# B&R Automation Studio project NewPendant_NG4_11_05_25A (part 18)

```c
					/////////////////////////
					/////   Hardcoded Limits
					if(cfg->HeadCfg.OSC.Limits_Harcoded){

						curCalib->Points[CALIB_OSC_SFT_LIMIT].num = 4;
						curCalib->Points[CALIB_OSC_SFT_LIMIT].val[0] = 10.0;
						curCalib->Points[CALIB_OSC_SFT_LIMIT].val[1] = 75.0;
						curCalib->Points[CALIB_OSC_SFT_LIMIT].val[2] = curCalib->Points[i].val[0];
						curCalib->Points[CALIB_OSC_SFT_LIMIT].val[3] = curCalib->Points[i].val[1];
					}

					////////////////////////////////////////////////

				break;

			}

		}

		for(i=0 ; i < 1 ; i++){

			switch(i){

				case 0:

					strcpy(Process[PROC_GAS].Name , "GAS");
					GAS_Param_Set[i].pPrc = &Process[PROC_GAS];

					//GAS_Param_Set[i].pSensInput     = &Hardware[1].Inp[5];  //FourAxis Head
					GAS_Param_Set[i].pOutput		= &Hardware[1].Outp[4];

				break;

			}

		}

		for(i=0 ; i < 1; i++){

			switch(i){

				case 0:

					strcpy(Process[PROC_COOL].Name , "COOLANT");
					COOL_Param_Set[i].pPrc = &Process[PROC_COOL];

					COOL_Param_Set[i].pSensInput     = &Hardware[1].Inp[4];  //FourAxis Head
					COOL_Param_Set[i].pOutput		= &Hardware[1].Outp[6];

				break;

			}

		}

		for(i=0 ; i < 1; i++){

			switch(i){

				case 0:

					strcpy(Process[PROC_HW_PS].Name , "HW PS");
					HW_PS_Param_Set[i].pPrc = &Process[PROC_HW_PS];

					HW_PS_Param_Set[i].pCalibPoints		= &m->pCalib->Points[CALIB_HW_AMPS_CMD];
					HW_PS_Param_Set[i].rawCmdMax 		= 16383.0;
					HW_PS_Param_Set[i].AmpCMD_Max 		= 160.0;

					Process[PROC_HW_PS].Disable = 1;

				break;

			}

		}

		for(i=0 ; i < 2; i++){

			switch(i){

				case 0:

					strcpy(Process[PROC_WIRE_FEED].Name ,"WrFeed");
					strcpy(VectorStateMach[VECT_WF].Name ,"WrFeed#1");
					strcpy(VectorStateMach[VECT_WF_1].Name ,"WrFeed#2");

					WIRE_Param_Set[i].pPrc = &Process[PROC_WIRE_FEED];
					WIRE_Param_Set[i].pVect = &VectorStateMach[m->pCfg->HeadCfg.WF.VECT_A_Indx];
					WIRE_Param_Set[i].VectStateNum = 1;
					WIRE_Param_Set[i].Mode = 0;  // classic

					WIRE_Param_Set[i].pCalibPoints	= &m->pCalib->Points[CALIB_WF_SPEED_CMD];

				break;

				case 1:

					strcpy(Process[PROC_WIRE_PULSE].Name ,"WrPulse");
					strcpy(VectorStateMach[VECT_WP].Name ,"WrPulse#1");
					strcpy(VectorStateMach[VECT_WP_1].Name ,"WrPulse#2");

					WIRE_Param_Set[i].pPrc = &Process[PROC_WIRE_PULSE];
					WIRE_Param_Set[i].pVect = &VectorStateMach[m->pCfg->HeadCfg.WP.VECT_A_Indx];
					WIRE_Param_Set[i].VectStateNum = 1;

					WIRE_Param_Set[i].pCalibPoints	= &m->pCalib->Points[CALIB_WP_SPEED_CMD];

					Process[PROC_WIRE_PULSE].Disable = 1;

				break;

		}

		}

		for(i=0 ; i < 1; i++){

			switch(i){

				case 0:

					strcpy(Process[PROC_TVL].Name , "TVL");
					strcpy(VectorStateMach[VECT_TVL].Name , "TVL");

					TVL_ROT_Param_Set[i].pPrc = &Process[PROC_TVL];
					TVL_ROT_Param_Set[i].pVect = &VectorStateMach[VECT_TVL];
					TVL_ROT_Param_Set[i].VectStateNum = 1;

					TVL_ROT_Param_Set[i].VectModeForJog = vectSt_Mode_Volt;

					TVL_ROT_Param_Set[i].MaxSpeedJog = 24.0;

					TVL_ROT_Param_Set[i].TotalRescaleFactor = 1.0;
					TVL_ROT_Param_Set[i].pCalibPoints = &m->pCalib->Points[CALIB_TVL_SPEED_CMD];

					TVL_ROT_Param_Set[i].pTrackDia = &curCfg->Param[parTVL_TrackDia].val[0];
					TVL_ROT_Param_Set[i].pVelTolerance = &curCfg->Param[parTVL_SpeedTolerane].val[0];

					TVL_ROT_Param_Set[i].pEncoder = &AxisCh[TML_AX_TVL].curPos;
					TVL_ROT_Param_Set[i].pHomePos = &OLD_MTR_POS[TVL_ENC_HOME];
					TVL_ROT_Param_Set[i].EncPerTick = m->pCfg->HeadCfg.TVL.EncPerTick;
					TVL_ROT_Param_Set[i].EncDir = m->pCfg->HeadCfg.TVL.Enc_Dir;
					TVL_ROT_Param_Set[i].TicksAtHighVel = 3;

				break;

			}
		}

		for(i=0 ; i < 1 ; i++){

			switch(i){

				case 0:

					strcpy(Process[m->pCfg->HeadCfg.INDX.PROC_Indx].Name , "INDX");
					INDEX_Param_Set[i].pPrc = &Process[m->pCfg->HeadCfg.INDX.PROC_Indx];
					Process[m->pCfg->HeadCfg.INDX.PROC_Indx].Disable = 1;

				break;

			}

		}

	return 1;

}

DINT Configure_F_HEAD_HP_MINI_ENC(MASTER_typ * m,UINT headType){
int i;

CurCfg_typ *curCfg;
Cfg_typ *cfg;
CurCalib_typ *curCalib , *defaultCalib;

	if(!m)
		return;

	curCfg = (CurCfg_typ*)m->pCurCfg;
	cfg = (Cfg_typ*)m->pCfg;

	curCalib = m->pCalib;
	defaultCalib = m->pDefaultCalib;

	if(!curCfg || !cfg || !curCalib  || !defaultCalib)
		return;

	/*********************************************/
	/***   Hardware and Vectors *********************/

	TML_MTR_INST[m->pCfg->HeadCfg.TVL.TML_Indx ].pState = &VectorStateMach[m->pCfg->HeadCfg.TVL.VECT_Indx];

	TML_MTR_INST[m->pCfg->HeadCfg.AVC.TML_A_Indx ].pState = &VectorStateMach[m->pCfg->HeadCfg.AVC.VECT_A_Indx];
	TML_MTR_INST[m->pCfg->HeadCfg.AVC.TML_B_Indx ].pState = &VectorStateMach[m->pCfg->HeadCfg.AVC.VECT_B_Indx];

	TML_MTR_INST[m->pCfg->HeadCfg.OSC.TML_A_Indx ].pState = &VectorStateMach[m->pCfg->HeadCfg.OSC.VECT_A_Indx];
	TML_MTR_INST[m->pCfg->HeadCfg.OSC.TML_B_Indx ].pState = &VectorStateMach[m->pCfg->HeadCfg.OSC.VECT_B_Indx];

	DC_Mtr[m->pCfg->HeadCfg.WF.DC_A_Indx ].pState = &VectorStateMach[m->pCfg->HeadCfg.WF.VECT_A_Indx];
	DC_Mtr[m->pCfg->HeadCfg.WP.DC_A_Indx ].pState = &VectorStateMach[m->pCfg->HeadCfg.WP.VECT_A_Indx];
	DC_Mtr[m->pCfg->HeadCfg.WF.DC_B_Indx ].pState = &VectorStateMach[m->pCfg->HeadCfg.WF.VECT_B_Indx];
	DC_Mtr[m->pCfg->HeadCfg.WP.DC_B_Indx ].pState = &VectorStateMach[m->pCfg->HeadCfg.WP.VECT_B_Indx];

/*

	VectorStateMach[VECT_AVC].simul = 1;
	VectorStateMach[VECT_OSC].simul = 1;
	VectorStateMach[VECT_TVL].simul = 1;
	VectorStateMach[VECT_WF].simul = 1;
	VectorStateMach[VECT_WP].simul = 1;
	VectorStateMach[VECT_WF_1].simul = 1;
	VectorStateMach[VECT_WP_1].simul = 1;
		m->pCfg->HeadCfg.WF.VECT_A_Indx]
	DC_Mtr[DC_AX_WF].Disable = 1;
	DC_Mtr[DC_AX_WP].Disable = 1;
	DC_Mtr[DC_AX_WF_1].Disable = 1;
	DC_Mtr[DC_AX_WP_1].Disable = 1;

	TML_MTR_INST[TML_AX_AVC].Disable = 1;
	TML_MTR_INST[TML_AX_OSC].Disable = 1;
	TML_MTR_INST[TML_AX_TVL].Disable = 1;

	//Process[PROC_AVC].Disable = 1;
	Process[PROC_AVC].TestMode = 1;
*/
	Process[PROC_TVL].Disable = 0;
	Process[PROC_OSC].Disable = 0;
	Process[PROC_AVC].Disable = 0;
	Process[PROC_WIRE_FEED].Disable = 0;
	Process[PROC_WIRE_PULSE].Disable = 0;

	VectorStateMach[VECT_AVC].simul = 0;
	VectorStateMach[VECT_OSC].simul = 0;
	VectorStateMach[VECT_TVL].simul = 0;

	DC_Mtr[DC_AX_WF].Disable = 0;
	DC_Mtr[DC_AX_WP].Disable = 0;
	DC_Mtr[DC_AX_WF_1].Disable = 1;
	DC_Mtr[DC_AX_WP_1].Disable = 1;

	TML_MTR_INST[TML_AX_AVC].Disable = 0;
	TML_MTR_INST[TML_AX_OSC].Disable = 0;
	TML_MTR_INST[TML_AX_TVL].Disable = 0;

	/*********************************************************/
	/****   Phisical hardware configuration   ************************/

		for(i = 0 ; i < PROCESS_NUM; i++)
			strcpy(Process[i].Name , "spare");

		for(i = 0 ; i < VECTORS_NUM; i++)
			strcpy(VectorStateMach[i].Name , "spare");

		//////////////////////////////////////////////////////////////////////////////////
		// Wire Block
		for(i=0 ; i < 2; i++){

			switch(i){

				case 0:
					strcpy(Process[m->pCfg->HeadCfg.WB[i].PROC_Indx].Name , "WB_UD");
					strcpy(VectorStateMach[m->pCfg->HeadCfg.WB[i].VECT_Indx].Name , "WB_UD");

					WR_BLK_Param_Set[i].pPrc = &Process[m->pCfg->HeadCfg.WB[i].PROC_Indx];
					WR_BLK_Param_Set[i].pVect = &VectorStateMach[m->pCfg->HeadCfg.WB[i].VECT_Indx];
					WR_BLK_Param_Set[i].VectStateNum = 1;

					WR_BLK_Param_Set[i].MaxSpeedJog = 24.0;

					Gen_one = 1.0;
					WR_BLK_Param_Set[i].pJogSpeed = &Gen_one;

				break;

				case 1:
					strcpy(Process[m->pCfg->HeadCfg.WB[i].PROC_Indx].Name , "WB_LR");
					strcpy(VectorStateMach[m->pCfg->HeadCfg.WB[i].VECT_Indx].Name , "WB_LR");

					WR_BLK_Param_Set[i].pPrc = &Process[PROC_WB_LR];
					WR_BLK_Param_Set[i].pVect = &VectorStateMach[VECT_WB_LR];
					WR_BLK_Param_Set[i].VectStateNum = 1;

					WR_BLK_Param_Set[i].MaxSpeedJog = 24.0;

					Gen_one = 1.0;
					WR_BLK_Param_Set[i].pJogSpeed = &Gen_one;

				break;

			}

		}

		for(i = 0 ; i < DC2DIRMTR_NUM; i++){

			switch(i){

				case DC_WB_UD:

					strcpy(DC2DirMtr[i].Name , "WB_UD");
					DC2DirMtr[i].pState = &VectorStateMach[VECT_WB_UD];

					DC2DirMtr[i].Cfg.pQ1_output = &Hardware[1].Outp[12];
					DC2DirMtr[i].Cfg.pQ2_output = &Hardware[1].Outp[13];
					DC2DirMtr[i].Cfg.pQ3_output = &Hardware[1].Outp[14];
					DC2DirMtr[i].Cfg.pQ4_output = &Hardware[1].Outp[15];

					DC2DirMtr[i].Cfg.MtrDir = 1.0;

				break;

				case DC_WB_LR:

					strcpy(DC2DirMtr[i].Name , "WB_LR");
					DC2DirMtr[i].pState = &VectorStateMach[VECT_WB_LR];

					DC2DirMtr[i].Cfg.pQ1_output = &Hardware[1].Outp[16];
					DC2DirMtr[i].Cfg.pQ2_output = &Hardware[1].Outp[17];
					DC2DirMtr[i].Cfg.pQ3_output = &Hardware[1].Outp[18];
					DC2DirMtr[i].Cfg.pQ4_output = &Hardware[1].Outp[19];

					DC2DirMtr[i].Cfg.MtrDir = 1.0;

				break;

			}

		}
		/////////////////////////////////////////////////////////////////////////////////

		for(i = 0 ; i < GEN_MTR_NUM; i++){

			switch(i){

				case DC_AX_WF:
				case DC_AX_WF_1:

					switch(i){

						case DC_AX_WF:

							strcpy(DC_Mtr[i].Name , "DC WFeed#1");

							DC_Mtr[i].Cfg.mtr_dir = 1.0;

							if(ProjectConfig == project_US_Orbital) // US Orbital has B and /B swapped
								DC_Mtr[i].Cfg.enc_dir = -1.0;
							else
								DC_Mtr[i].Cfg.enc_dir = 1.0;

						break;

						case DC_AX_WF_1:

							strcpy(DC_Mtr[i].Name , "DC WFeed#2");

							//DC_Mtr[i].Cfg.mtr_dir = -1.0;
							DC_Mtr[i].Cfg.mtr_dir = 1.0;

							if(ProjectConfig == project_US_Orbital) // US Orbital has B and /B swapped
								DC_Mtr[i].Cfg.enc_dir = -1.0;
							else
								DC_Mtr[i].Cfg.enc_dir = 1.0;

						break;

					}

					//DC_Mtr[i].Cfg.units = 59.847340050885561192713356451475; // 0.75 " dia * 25.4 * PI
					DC_Mtr[i].Cfg.units = 2000 / 59.847340050885561192713356451475; // 2000 enc ticks / 0.75 " dia * 25.4 * PI
					DC_Mtr[i].Cfg.rev_scale = 66.0;	// Ratio gear box 66:1

					/* Parameters for PID controller */
					// To nowe
					DC_Mtr[i].msc.PIDParameters.Kp= 1.0;//0.4; //proportional gain / was 0.6
					//DC_Mtr[i].msc.PIDParameters.Kp= 0.1;//0.4; //proportional gain / was 0.6
					DC_Mtr[i].msc.PIDParameters.Tn= 0.1;//0.3.1; //intergral action time
					DC_Mtr[i].msc.PIDParameters.Kfbk = 0.01; //windup dampenin

					DC_Mtr[i].msc.PID.enable = 0;
					DC_Mtr[i].msc.PID.pPar = &DC_Mtr[i].msc.PIDParameters;
					DC_Mtr[i].msc.PID.request = 3; // Read parameters from PIDParameters
					DC_Mtr[i].msc.PIDParameters.Tv= 0; //derivative action time
					DC_Mtr[i].msc.PIDParameters.Y_max = 100.0;  //max manipulated variable %
					DC_Mtr[i].msc.PIDParameters.Y_min = -100.0; //min manipulated variable %

				break;

				case DC_AX_WP:
				case DC_AX_WP_1:

					switch(i){

						case DC_AX_WP:

							strcpy(DC_Mtr[i].Name , "DC WPulse#1");

							DC_Mtr[i].Cfg.mtr_dir = 1.0;

							if(ProjectConfig == project_US_Orbital) // US Orbital has B and /B swapped
								DC_Mtr[i].Cfg.enc_dir = -1.0;
							else
								DC_Mtr[i].Cfg.enc_dir = 1.0;

						break;

						case DC_AX_WP_1:

							strcpy(DC_Mtr[i].Name , "DC WPulse#2");

							DC_Mtr[i].Cfg.mtr_dir = 1.0;

							if(ProjectConfig == project_US_Orbital) // US Orbital has B and /B swapped
								DC_Mtr[i].Cfg.enc_dir = -1.0;
							else
								DC_Mtr[i].Cfg.enc_dir = 1.0;

						break;

					}

					//oryginalnie jest 2000 pulsow na obrot potem ratio on gear 4.8 : 1
					DC_Mtr[i].Cfg.units = 2000;
					DC_Mtr[i].Cfg.rev_scale = 4.8;// ratio on gear 4.8

					/* Parameters for PID controller */
					// To nowe
					DC_Mtr[i].msc.PIDParameters.Kp= 1.0;//0.4; //proportional gain / was 0.6
					//DC_Mtr[i].msc.PIDParameters.Kp= 0.1;//0.4; //proportional gain / was 0.6
					DC_Mtr[i].msc.PIDParameters.Tn= 0.1;//0.3.1; //intergral action time
					DC_Mtr[i].msc.PIDParameters.Kfbk = 0.01; //windup dampenin

					DC_Mtr[i].msc.PID.enable = 0;
					DC_Mtr[i].msc.PID.pPar = &DC_Mtr[i].msc.PIDParameters;
					DC_Mtr[i].msc.PID.request = 3; // Read parameters from PIDParameters
					DC_Mtr[i].msc.PIDParameters.Tv= 0; //derivative action time
					DC_Mtr[i].msc.PIDParameters.Y_max = 100.0;  //max manipulated variable %
					DC_Mtr[i].msc.PIDParameters.Y_min = -100.0; //min manipulated variable %

				break;

				default:

					strcpy(DC_Mtr[i].Name , "Spare ");

				break;

			}

			//CalcUnits(&DC_Mtr[i]);
			DC_Mtr[i].msc.kPos = (float)DC_Mtr[i].Cfg.units * DC_Mtr[i].Cfg.rev_scale;

		}

		/***********************************/

			for(i = 0 ; i < TML_SERVO_NUM ; i++){

				switch(i){

					// tml->_int.kPos = (tml->_cfg.units * tml->_cfg.rev_scale) / tml->_cfg.rev_motor;
					case TML_AX_AVC:

						strcpy(TML_MTR_INST[i].Name , "AVC");

						// Analog Feedback from REF
						TML_MTR_INST[i]._cfg.loopPeriod = 0.001;
						TML_MTR_INST[i]._cfg.units = 4095;
						TML_MTR_INST[i]._cfg.rev_motor = 1;
						TML_MTR_INST[i]._cfg.rev_scale = 1.0/5.0;
						TML_MTR_INST[i]._cfg.maxVel = 10.0; //1//6000 rpm
						TML_MTR_INST[i]._cfg.maxAcc = 100000.0;
						//TML_MTR_INST[i]._cfg.satpMax = 27853; // KPP bylo Stauration of proportional gain
						TML_MTR_INST[i]._cfg.satpMax = 32000; // KPP bylo Stauration of proportional gain
						TML_MTR_INST[i]._cfg.kppMax = 32000; // KPP bylo Stauration of proportional gain
						TML_MTR_INST[i]._cfg.kipMax = 200; // KPP bylo Stauration of proportional gain
						TML_MTR_INST[i]._cfg.absFbk = 0; // absolute value feedback

						TML_MTR_INST[i]._cfg.signFilter = curCfg->Param[parAVC_FbkFilter].val[0];

						if(ProjectConfig == project_US_Orbital){
							strcpy(TML_MTR_INST[i]._cfg.programName , "1423_AVC_FH_MINI_ENC_US.sw");
							TML_MTR_INST[i].ProgramVersion = ASC2UDINT("1423");
							TML_MTR_INST[i].FirmwareVersion = ASC2UDINT("6A2B");  //0x674B
							TML_MTR_INST[i]._cfg.Appl_ID_adr = 0x7FCF;

						}
						else{
							strcpy(TML_MTR_INST[i]._cfg.programName , "0423_AVC_FH_MINI_ENC.sw");
							TML_MTR_INST[i].ProgramVersion = ASC2UDINT("0423");
							TML_MTR_INST[i].FirmwareVersion = ASC2UDINT("674C");  //0x674C
						}

						//TML_MTR_INST[i]._cfg.sftLimitPos = 1000.0;
						//TML_MTR_INST[i]._cfg.sftLimitNeg = -1000.0;

					break;

					case TML_AX_OSC:

						strcpy(TML_MTR_INST[i].Name , "OSC");

						if(ProjectConfig == project_US_Orbital){
							strcpy(TML_MTR_INST[i]._cfg.programName , "1412_OSC_FH_MINI_ENC_US.sw");
							TML_MTR_INST[i].ProgramVersion = ASC2UDINT("1412");
							TML_MTR_INST[i].FirmwareVersion = ASC2UDINT("6A2B");  //0x674B
							TML_MTR_INST[i]._cfg.Appl_ID_adr = 0x7FCF;

						}
						else{
							strcpy(TML_MTR_INST[i]._cfg.programName , "0412_OSC_FH_MINI_ENC.sw");
							TML_MTR_INST[i].ProgramVersion = ASC2UDINT("0412");
							TML_MTR_INST[i].FirmwareVersion = ASC2UDINT("674C");  //0x674C
						}

						TML_MTR_INST[i]._cfg.loopPeriod = 0.001;
						TML_MTR_INST[i]._cfg.absFbk = 0; // value fom APOS which is analog Ref
						TML_MTR_INST[i]._cfg.units = 4096.0 ;
						TML_MTR_INST[i]._cfg.rev_motor = 1;
						TML_MTR_INST[i]._cfg.rev_scale = 1.0 / 80.0;  // this comes from experiment
						//TML_MTR_INST[i]._cfg.rev_scale = 1.0 / 56.0; // this comes from drawings
						TML_MTR_INST[i]._cfg.maxVel = 100.0;
						TML_MTR_INST[i]._cfg.maxAcc = 100.0;

						TML_MTR_INST[i]._cfg.AnalLimitPos = 3900;
						TML_MTR_INST[i]._cfg.AnalLimitNeg = 100;

					break;

					case TML_AX_TVL:

						strcpy(TML_MTR_INST[i].Name , "TVL");

						/// Deferent TML programs
						// Back EMF
						TML_MTR_INST[i]._cfg.loopPeriod = 0.001;

						if(ProjectConfig == project_US_Orbital){
							strcpy(TML_MTR_INST[i]._cfg.programName , "1411_TVL_FH_MINI_ENC_US.sw");
							TML_MTR_INST[i].ProgramVersion = ASC2UDINT("1411");
							TML_MTR_INST[i].FirmwareVersion = ASC2UDINT("6A2B");  //0x674B
							TML_MTR_INST[i]._cfg.Appl_ID_adr = 0x7FCF;

						}
						else{
							strcpy(TML_MTR_INST[i]._cfg.programName , "0411_TVL_FH_MINI_ENC.sw");
							TML_MTR_INST[i].ProgramVersion = ASC2UDINT("0411");
							TML_MTR_INST[i].FirmwareVersion = ASC2UDINT("674C");  //0x674C
						}

						TML_MTR_INST[i]._cfg.units =  1000; //  to jest tyle ile z max speed TML EREF
						TML_MTR_INST[i]._cfg.rev_scale = -1920.0;
						TML_MTR_INST[i]._cfg.rev_motor = 1.0 ;
						TML_MTR_INST[i]._cfg.maxVel =  10.0; // mm/s
						TML_MTR_INST[i]._cfg.maxAcc = 100.0;
						TML_MTR_INST[i]._cfg.absFbk = 0; // non absolute value feedback , remember last value before drive reset

					break;

					default:

						xsprintf(TML_MTR_INST[i].Name, "Spare %d", i );
						TML_MTR_INST[i].pState = 0;

					break;

				}

			TML_MTR_INST[i].xCMD = TML_RESTART;

		}

		TML_mgr[0].hrdw[0].AxisNum = 3;
		TML_mgr[0].hrdw[1].AxisNum = 0;

		TML_mgr[0].pAxis[0] = &AxisCh[0];
		TML_mgr[0].pAxis[1] = 0;
		//TML_mgr[0].pAxis[1] = &AxisCh[TML_mgr[0].hrdw[0].AxisNum];

		TML_mgr[0].pTML[0] = &TML_MTR_INST[0];
		TML_mgr[0].pTML[1] = 0;
		//TML_mgr[0].pTML[1] = &TML_MTR_INST[TML_mgr[0].hrdw[0].AxisNum];

		AxisCh[TML_AX_TVL].AxisID	= 1;
		AxisCh[TML_AX_OSC].AxisID 	= 2;
		AxisCh[TML_AX_AVC].AxisID 	= 3;

		/**************************************/
		/****   Process   ************************/

		// Lincoln Power Supply
		for(i=0 ; i < 1; i++){

			switch(i){

				case 0:

					strcpy(Process[PROC_TIG_PS].Name , "TIG PS");
					PS_Param_Set[i].pPrc = &Process[PROC_TIG_PS];

					PS_Param_Set[i].pCalibPoints		= &m->pCalib->Points[CALIB_TIG_AMPS_CMD];
					//PS_Param_Set[i].rawCmdMax			= 26170; // //
					//PS_Param_Set[i].AmpCMD_Max			= 500.0; // 62.5 amp / 1 V
					PS_Param_Set[i].rawCmdMax			= 32767;
					PS_Param_Set[i].AmpCMD_Max			= 627.0;

					PS_Param_Set[i].pArcLinkRobot   = (UDINT)&ArcLink.robot;

				break;

			}

		}

		for(i=0 ; i < 1 ; i++){

			switch(i){

				case 0:

					strcpy(Process[PROC_AVC].Name , "AVC");

					strcpy(VectorStateMach[VECT_AVC].Name , "AVC");

					AVC_Param_Set[i].pPrc = &Process[PROC_AVC];
					AVC_Param_Set[i].pVect = &VectorStateMach[VECT_AVC];
					AVC_Param_Set[i].VectStateNum = 1;
					AVC_Param_Set[i].Mode = 0;

					AVC_Param_Set[i].MaxSpeedJog = 24.0;

					m->pCalib->Points[CALIB_TIG_VOLT_FBK].num = 10;
					AVC_Param_Set[i].pCalibPoints		= &m->pCalib->Points[CALIB_TIG_VOLT_FBK];

				break;

			}
		}

		for(i=0 ; i < 1 ; i++){

			switch(i){

				case 0:

					strcpy(Process[PROC_OSC].Name , "OSC");
					strcpy(VectorStateMach[VECT_OSC].Name , "OSC");

					OSC_TML_Param_Set[i].pPrc = &Process[PROC_OSC];
					OSC_TML_Param_Set[i].pVect = &VectorStateMach[VECT_OSC];
					OSC_TML_Param_Set[i].VectStateNum = 1;
					OSC_TML_Param_Set[i].pTML = &TML_MTR_INST[TML_AX_OSC] ;

					OSC_TML_Param_Set[i].Mode = 0;

					////  New Oscillation concept - BEMF
					OSC_TML_Param_Set[i].mm2ticks = TML_MTR_INST[TML_AX_OSC]._cfg.units * TML_MTR_INST[TML_AX_OSC]._cfg.rev_scale;
			 		OSC_TML_Param_Set[i].SpeedFactor = 410;
					//OSC_TML_Param_Set[i].MaxOscAmpl = 1.0 * 25.4;
					OSC_TML_Param_Set[i].MaxOscAmpl = 0.0;

					/////////////////////////
					/////   Hardcoded Limits
					if(cfg->HeadCfg.OSC.Limits_Harcoded){

						curCalib->Points[CALIB_OSC_SFT_LIMIT].num = 4;
						curCalib->Points[CALIB_OSC_SFT_LIMIT].val[0] = 10.0;
						curCalib->Points[CALIB_OSC_SFT_LIMIT].val[1] = 75.0;
						curCalib->Points[CALIB_OSC_SFT_LIMIT].val[2] = curCalib->Points[i].val[0];
						curCalib->Points[CALIB_OSC_SFT_LIMIT].val[3] = curCalib->Points[i].val[1];
					}

					////////////////////////////////////////////////

				break;

			}

		}

		for(i=0 ; i < 1 ; i++){

			switch(i){

				case 0:

					strcpy(Process[PROC_GAS].Name , "GAS");
					GAS_Param_Set[i].pPrc = &Process[PROC_GAS];

					//GAS_Param_Set[i].pSensInput     = &Hardware[1].Inp[5];  //FourAxis Head
					GAS_Param_Set[i].pOutput		= &Hardware[1].Outp[4];

				break;

			}

		}

		for(i=0 ; i < 1; i++){

			switch(i){

				case 0:

					strcpy(Process[PROC_COOL].Name , "COOLANT");
					COOL_Param_Set[i].pPrc = &Process[PROC_COOL];

					COOL_Param_Set[i].pSensInput     = &Hardware[1].Inp[4];  //FourAxis Head
					COOL_Param_Set[i].pOutput		= &Hardware[1].Outp[6];

				break;

			}

		}

		for(i=0 ; i < 1; i++){

			switch(i){

				case 0:

					strcpy(Process[PROC_HW_PS].Name , "HW PS");
					HW_PS_Param_Set[i].pPrc = &Process[PROC_HW_PS];

					HW_PS_Param_Set[i].pCalibPoints		= &m->pCalib->Points[CALIB_HW_AMPS_CMD];
					HW_PS_Param_Set[i].rawCmdMax 		= 16383.0;
					HW_PS_Param_Set[i].AmpCMD_Max 		= 160.0;

				break;

			}

		}

		for(i=0 ; i < 2; i++){

			switch(i){

				case 0:

					strcpy(Process[PROC_WIRE_FEED].Name ,"WrFeed");
					strcpy(VectorStateMach[VECT_WF].Name ,"WrFeed#1");
					strcpy(VectorStateMach[VECT_WF_1].Name ,"WrFeed#2");

					WIRE_Param_Set[i].pPrc = &Process[PROC_WIRE_FEED];
					WIRE_Param_Set[i].pVect = &VectorStateMach[m->pCfg->HeadCfg.WF.VECT_A_Indx];
					WIRE_Param_Set[i].VectStateNum = 1;
					WIRE_Param_Set[i].Mode = 0;  // classic

					WIRE_Param_Set[i].pCalibPoints	= &m->pCalib->Points[CALIB_WF_SPEED_CMD];

				break;

				case 1:

					strcpy(Process[PROC_WIRE_PULSE].Name ,"WrPulse");
					strcpy(VectorStateMach[VECT_WP].Name ,"WrPulse#1");
					strcpy(VectorStateMach[VECT_WP_1].Name ,"WrPulse#2");

					WIRE_Param_Set[i].pPrc = &Process[PROC_WIRE_PULSE];
					WIRE_Param_Set[i].pVect = &VectorStateMach[m->pCfg->HeadCfg.WP.VECT_A_Indx];
					WIRE_Param_Set[i].VectStateNum = 1;

					WIRE_Param_Set[i].pCalibPoints	= &m->pCalib->Points[CALIB_WP_SPEED_CMD];

				break;

		}

		}

		for(i=0 ; i < 1; i++){

			switch(i){

				case 0:

					strcpy(Process[PROC_TVL].Name , "TVL");
					strcpy(VectorStateMach[VECT_TVL].Name , "TVL");

					TVL_ROT_Param_Set[i].pPrc = &Process[PROC_TVL];
					TVL_ROT_Param_Set[i].pVect = &VectorStateMach[VECT_TVL];
					TVL_ROT_Param_Set[i].VectStateNum = 1;

					TVL_ROT_Param_Set[i].VectModeForJog = vectSt_Mode_Volt;

					TVL_ROT_Param_Set[i].MaxSpeedJog = 24.0;

					TVL_ROT_Param_Set[i].TotalRescaleFactor = 1.0;
					TVL_ROT_Param_Set[i].pCalibPoints = &m->pCalib->Points[CALIB_TVL_SPEED_CMD];

					TVL_ROT_Param_Set[i].pTrackDia = &curCfg->Param[parTVL_TrackDia].val[0];
					TVL_ROT_Param_Set[i].pVelTolerance = &curCfg->Param[parTVL_SpeedTolerane].val[0];

					TVL_ROT_Param_Set[i].pEncoder = &AxisCh[TML_AX_TVL].curPos;
					TVL_ROT_Param_Set[i].pHomePos = &OLD_MTR_POS[TVL_ENC_HOME];
					TVL_ROT_Param_Set[i].EncPerTick = m->pCfg->HeadCfg.TVL.EncPerTick;
					TVL_ROT_Param_Set[i].EncDir = m->pCfg->HeadCfg.TVL.Enc_Dir;
					TVL_ROT_Param_Set[i].TicksAtHighVel = 3;

				break;

			}
		}

		for(i=0 ; i < 1 ; i++){

			switch(i){

				case 0:

					strcpy(Process[m->pCfg->HeadCfg.INDX.PROC_Indx].Name , "INDX");
					INDEX_Param_Set[i].pPrc = &Process[m->pCfg->HeadCfg.INDX.PROC_Indx];
					Process[m->pCfg->HeadCfg.INDX.PROC_Indx].Disable = 1;

				break;

			}

		}

	return 1;

}

DINT Configure_D_HEAD_HP(MASTER_typ * m,UINT headType){
int i;

CurCfg_typ *curCfg;
Cfg_typ *cfg;
CurCalib_typ *curCalib , *defaultCalib;

	if(!m)
		return;

	curCfg = (CurCfg_typ*)m->pCurCfg;
	cfg = (Cfg_typ*)m->pCfg;

	curCalib = m->pCalib;
	defaultCalib = m->pDefaultCalib;

	if(!curCfg || !cfg || !curCalib  || !defaultCalib)
		return;

	/*********************************************/
	/***   Hardware and Vectors *********************/

	TML_MTR_INST[m->pCfg->HeadCfg.TVL.TML_Indx ].pState = &VectorStateMach[m->pCfg->HeadCfg.TVL.VECT_Indx];

	TML_MTR_INST[m->pCfg->HeadCfg.AVC.TML_A_Indx ].pState = &VectorStateMach[m->pCfg->HeadCfg.AVC.VECT_A_Indx];
	TML_MTR_INST[m->pCfg->HeadCfg.AVC.TML_B_Indx ].pState = &VectorStateMach[m->pCfg->HeadCfg.AVC.VECT_B_Indx];

	TML_MTR_INST[m->pCfg->HeadCfg.OSC.TML_A_Indx ].pState = &VectorStateMach[m->pCfg->HeadCfg.OSC.VECT_A_Indx];
	TML_MTR_INST[m->pCfg->HeadCfg.OSC.TML_B_Indx ].pState = &VectorStateMach[m->pCfg->HeadCfg.OSC.VECT_B_Indx];

	DC_Mtr[m->pCfg->HeadCfg.WF.DC_A_Indx ].pState = &VectorStateMach[m->pCfg->HeadCfg.WF.VECT_A_Indx];
	DC_Mtr[m->pCfg->HeadCfg.WP.DC_A_Indx ].pState = &VectorStateMach[m->pCfg->HeadCfg.WP.VECT_A_Indx];
	DC_Mtr[m->pCfg->HeadCfg.WF.DC_B_Indx ].pState = &VectorStateMach[m->pCfg->HeadCfg.WF.VECT_B_Indx];
	DC_Mtr[m->pCfg->HeadCfg.WP.DC_B_Indx ].pState = &VectorStateMach[m->pCfg->HeadCfg.WP.VECT_B_Indx];

/*

	VectorStateMach[VECT_AVC].simul = 1;
	VectorStateMach[VECT_OSC].simul = 1;
	VectorStateMach[VECT_TVL].simul = 1;
	VectorStateMach[VECT_WF].simul = 1;
	VectorStateMach[VECT_WP].simul = 1;
	VectorStateMach[VECT_WF_1].simul = 1;
	VectorStateMach[VECT_WP_1].simul = 1;
		m->pCfg->HeadCfg.WF.VECT_A_Indx]
	DC_Mtr[DC_AX_WF].Disable = 1;
	DC_Mtr[DC_AX_WP].Disable = 1;
	DC_Mtr[DC_AX_WF_1].Disable = 1;
	DC_Mtr[DC_AX_WP_1].Disable = 1;

	TML_MTR_INST[TML_AX_AVC].Disable = 1;
	TML_MTR_INST[TML_AX_OSC].Disable = 1;
	TML_MTR_INST[TML_AX_TVL].Disable = 1;

	//Process[PROC_AVC].Disable = 1;
	Process[PROC_AVC].TestMode = 1;
*/
	Process[PROC_TVL].Disable = 0;
	Process[PROC_OSC].Disable = 0;
	Process[PROC_AVC].Disable = 0;
	Process[PROC_WIRE_FEED].Disable = 0;
	Process[PROC_WIRE_PULSE].Disable = 0;

	VectorStateMach[VECT_AVC].simul = 0;
	VectorStateMach[VECT_OSC].simul = 0;
	VectorStateMach[VECT_TVL].simul = 0;

	DC_Mtr[DC_AX_WF].Disable = 0;
	DC_Mtr[DC_AX_WP].Disable = 0;
	DC_Mtr[DC_AX_WF_1].Disable = 1;
	DC_Mtr[DC_AX_WP_1].Disable = 1;

	TML_MTR_INST[TML_AX_AVC].Disable = 0;
	TML_MTR_INST[TML_AX_OSC].Disable = 0;
	TML_MTR_INST[TML_AX_TVL].Disable = 0;

	/*********************************************************/
	/****   Phisical hardware configuration   ************************/

		for(i = 0 ; i < PROCESS_NUM; i++)
			strcpy(Process[i].Name , "spare");

		for(i = 0 ; i < VECTORS_NUM; i++)
			strcpy(VectorStateMach[i].Name , "spare");

		//////////////////////////////////////////////////////////////////////////////////
		// Wire Block
		for(i=0 ; i < 2; i++){

			switch(i){

				case 0:
					strcpy(Process[m->pCfg->HeadCfg.WB[i].PROC_Indx].Name , "WB_UD");
					strcpy(VectorStateMach[m->pCfg->HeadCfg.WB[i].VECT_Indx].Name , "WB_UD");

					WR_BLK_Param_Set[i].pPrc = &Process[m->pCfg->HeadCfg.WB[i].PROC_Indx];
					WR_BLK_Param_Set[i].pVect = &VectorStateMach[m->pCfg->HeadCfg.WB[i].VECT_Indx];
					WR_BLK_Param_Set[i].VectStateNum = 1;

					WR_BLK_Param_Set[i].MaxSpeedJog = 24.0;

					Gen_one = 1.0;
					WR_BLK_Param_Set[i].pJogSpeed = &Gen_one;

				break;

				case 1:
					strcpy(Process[m->pCfg->HeadCfg.WB[i].PROC_Indx].Name , "WB_LR");
					strcpy(VectorStateMach[m->pCfg->HeadCfg.WB[i].VECT_Indx].Name , "WB_LR");

					WR_BLK_Param_Set[i].pPrc = &Process[PROC_WB_LR];
					WR_BLK_Param_Set[i].pVect = &VectorStateMach[VECT_WB_LR];
					WR_BLK_Param_Set[i].VectStateNum = 1;

					WR_BLK_Param_Set[i].MaxSpeedJog = 24.0;

					Gen_one = 1.0;
					WR_BLK_Param_Set[i].pJogSpeed = &Gen_one;

				break;

			}

		}

		for(i = 0 ; i < DC2DIRMTR_NUM; i++){

			switch(i){

				case DC_WB_UD:

					strcpy(DC2DirMtr[i].Name , "WB_UD");
					DC2DirMtr[i].pState = &VectorStateMach[VECT_WB_UD];

					DC2DirMtr[i].Cfg.pQ1_output = &Hardware[1].Outp[12];
					DC2DirMtr[i].Cfg.pQ2_output = &Hardware[1].Outp[13];
					DC2DirMtr[i].Cfg.pQ3_output = &Hardware[1].Outp[14];
					DC2DirMtr[i].Cfg.pQ4_output = &Hardware[1].Outp[15];

					DC2DirMtr[i].Cfg.MtrDir = 1.0;

				break;

				case DC_WB_LR:

					strcpy(DC2DirMtr[i].Name , "WB_LR");
					DC2DirMtr[i].pState = &VectorStateMach[VECT_WB_LR];

					DC2DirMtr[i].Cfg.pQ1_output = &Hardware[1].Outp[16];
					DC2DirMtr[i].Cfg.pQ2_output = &Hardware[1].Outp[17];
					DC2DirMtr[i].Cfg.pQ3_output = &Hardware[1].Outp[18];
					DC2DirMtr[i].Cfg.pQ4_output = &Hardware[1].Outp[19];

					DC2DirMtr[i].Cfg.MtrDir = 1.0;

				break;

			}

		}
		/////////////////////////////////////////////////////////////////////////////////

		for(i = 0 ; i < GEN_MTR_NUM; i++){

			switch(i){

				case DC_AX_WF:
				case DC_AX_WF_1:

					switch(i){

						case DC_AX_WF:

							strcpy(DC_Mtr[i].Name , "DC WFeed#1");

							DC_Mtr[i].Cfg.mtr_dir = 1.0;

							if(ProjectConfig == project_US_Orbital) // US Orbital has B and /B swapped
								DC_Mtr[i].Cfg.enc_dir = -1.0;
							else
								DC_Mtr[i].Cfg.enc_dir = 1.0;

						break;

						case DC_AX_WF_1:

							strcpy(DC_Mtr[i].Name , "DC WFeed#2");

							//DC_Mtr[i].Cfg.mtr_dir = -1.0;
							DC_Mtr[i].Cfg.mtr_dir = 1.0;

							if(ProjectConfig == project_US_Orbital) // US Orbital has B and /B swapped
								DC_Mtr[i].Cfg.enc_dir = -1.0;
							else
								DC_Mtr[i].Cfg.enc_dir = 1.0;

						break;

					}

					//DC_Mtr[i].Cfg.units = 59.847340050885561192713356451475; // 0.75 " dia * 25.4 * PI
					DC_Mtr[i].Cfg.units = 2000 / 59.847340050885561192713356451475; // 2000 enc ticks / 0.75 " dia * 25.4 * PI
					DC_Mtr[i].Cfg.rev_scale = 66.0;	// Ratio gear box 66:1

					/* Parameters for PID controller */
					// To nowe
					DC_Mtr[i].msc.PIDParameters.Kp= 1.0;//0.4; //proportional gain / was 0.6
					//DC_Mtr[i].msc.PIDParameters.Kp= 0.1;//0.4; //proportional gain / was 0.6
					DC_Mtr[i].msc.PIDParameters.Tn= 0.1;//0.3.1; //intergral action time
					DC_Mtr[i].msc.PIDParameters.Kfbk = 0.01; //windup dampenin

					DC_Mtr[i].msc.PID.enable = 0;
					DC_Mtr[i].msc.PID.pPar = &DC_Mtr[i].msc.PIDParameters;
					DC_Mtr[i].msc.PID.request = 3; // Read parameters from PIDParameters
					DC_Mtr[i].msc.PIDParameters.Tv= 0; //derivative action time
					DC_Mtr[i].msc.PIDParameters.Y_max = 100.0;  //max manipulated variable %
					DC_Mtr[i].msc.PIDParameters.Y_min = -100.0; //min manipulated variable %

				break;

				case DC_AX_WP:
				case DC_AX_WP_1:

					switch(i){

						case DC_AX_WP:

							strcpy(DC_Mtr[i].Name , "DC WPulse#1");

							DC_Mtr[i].Cfg.mtr_dir = 1.0;

							if(ProjectConfig == project_US_Orbital) // US Orbital has B and /B swapped
								DC_Mtr[i].Cfg.enc_dir = -1.0;
							else
								DC_Mtr[i].Cfg.enc_dir = 1.0;

						break;

						case DC_AX_WP_1:

							strcpy(DC_Mtr[i].Name , "DC WPulse#2");

							DC_Mtr[i].Cfg.mtr_dir = 1.0;

							if(ProjectConfig == project_US_Orbital) // US Orbital has B and /B swapped
								DC_Mtr[i].Cfg.enc_dir = -1.0;
							else
								DC_Mtr[i].Cfg.enc_dir = 1.0;

						break;

					}

					//oryginalnie jest 2000 pulsow na obrot potem ratio on gear 4.8 : 1
					DC_Mtr[i].Cfg.units = 2000;
					DC_Mtr[i].Cfg.rev_scale = 4.8;// ratio on gear 4.8

					/* Parameters for PID controller */
					// To nowe
					DC_Mtr[i].msc.PIDParameters.Kp= 1.0;//0.4; //proportional gain / was 0.6
					//DC_Mtr[i].msc.PIDParameters.Kp= 0.1;//0.4; //proportional gain / was 0.6
					DC_Mtr[i].msc.PIDParameters.Tn= 0.1;//0.3.1; //intergral action time
					DC_Mtr[i].msc.PIDParameters.Kfbk = 0.01; //windup dampenin

					DC_Mtr[i].msc.PID.enable = 0;
					DC_Mtr[i].msc.PID.pPar = &DC_Mtr[i].msc.PIDParameters;
					DC_Mtr[i].msc.PID.request = 3; // Read parameters from PIDParameters
					DC_Mtr[i].msc.PIDParameters.Tv= 0; //derivative action time
					DC_Mtr[i].msc.PIDParameters.Y_max = 100.0;  //max manipulated variable %
					DC_Mtr[i].msc.PIDParameters.Y_min = -100.0; //min manipulated variable %

				break;

				default:

					strcpy(DC_Mtr[i].Name , "Spare ");

				break;

			}

			//CalcUnits(&DC_Mtr[i]);
			DC_Mtr[i].msc.kPos = (float)DC_Mtr[i].Cfg.units * DC_Mtr[i].Cfg.rev_scale;

		}

		/***********************************/

			for(i = 0 ; i < TML_SERVO_NUM ; i++){

				switch(i){

					// tml->_int.kPos = (tml->_cfg.units * tml->_cfg.rev_scale) / tml->_cfg.rev_motor;
					case TML_AX_AVC:

						strcpy(TML_MTR_INST[i].Name , "AVC");

						// Analog Feedback from REF
						TML_MTR_INST[i]._cfg.loopPeriod = 0.001;
						TML_MTR_INST[i]._cfg.units = 4095;
						TML_MTR_INST[i]._cfg.rev_motor = -1;
						TML_MTR_INST[i]._cfg.rev_scale = 1.0/5.0;
						TML_MTR_INST[i]._cfg.maxVel = 10.0; //1//6000 rpm
						TML_MTR_INST[i]._cfg.maxAcc = 100000.0;
						//TML_MTR_INST[i]._cfg.satpMax = 27853; // KPP bylo Stauration of proportional gain
						TML_MTR_INST[i]._cfg.satpMax = 32000; // KPP bylo Stauration of proportional gain
						TML_MTR_INST[i]._cfg.kppMax = 32000; // KPP bylo Stauration of proportional gain
						TML_MTR_INST[i]._cfg.kipMax = 200; // KPP bylo Stauration of proportional gain
						TML_MTR_INST[i]._cfg.absFbk = 0; // absolute value feedback

						TML_MTR_INST[i]._cfg.signFilter = curCfg->Param[parAVC_FbkFilter].val[0];

						if(ProjectConfig == project_US_Orbital){

							strcpy(TML_MTR_INST[i]._cfg.programName , "1423_AVC_FH_MINI_ENC_US.sw");
							TML_MTR_INST[i].ProgramVersion = ASC2UDINT("1423");
							TML_MTR_INST[i].FirmwareVersion = ASC2UDINT("6A2B");  //0x674B
							TML_MTR_INST[i]._cfg.Appl_ID_adr = 0x7FCF;

						}
						else{
							strcpy(TML_MTR_INST[i]._cfg.programName , "0423_AVC_FH_MINI_ENC.sw");
							TML_MTR_INST[i].ProgramVersion = ASC2UDINT("0423");
							TML_MTR_INST[i].FirmwareVersion = ASC2UDINT("674C");  //0x674C
						}

						//TML_MTR_INST[i]._cfg.sftLimitPos = 1000.0;
						//TML_MTR_INST[i]._cfg.sftLimitNeg = -1000.0;

					break;

					case TML_AX_OSC:

						strcpy(TML_MTR_INST[i].Name , "OSC");

						if(ProjectConfig == project_US_Orbital){

							/*
							strcpy(TML_MTR_INST[i]._cfg.programName , "1412_OSC_FH_MINI_ENC_US.sw");
							TML_MTR_INST[i].ProgramVersion = ASC2UDINT("1412");
							TML_MTR_INST[i].FirmwareVersion = ASC2UDINT("6A2B");  //0x674B
							TML_MTR_INST[i]._cfg.Appl_ID_adr = 0x7FCF;
							*/

							// New Osc Mode -  11;
							strcpy(TML_MTR_INST[i]._cfg.programName , "2512_OSC_D_HEAD_US.sw");
							TML_MTR_INST[i].ProgramVersion = ASC2UDINT("2512");
							TML_MTR_INST[i].FirmwareVersion = ASC2UDINT("6A2B");  //0x674B
							TML_MTR_INST[i]._cfg.Appl_ID_adr = 0x7FCF;

						}
						else{
							strcpy(TML_MTR_INST[i]._cfg.programName , "0412_OSC_FH_MINI_ENC.sw");
							TML_MTR_INST[i].ProgramVersion = ASC2UDINT("0412");
							TML_MTR_INST[i].FirmwareVersion = ASC2UDINT("674C");  //0x674C
						}

						TML_MTR_INST[i]._cfg.loopPeriod = 0.001;
						TML_MTR_INST[i]._cfg.absFbk = 0; // value fom APOS which is analog Ref
						TML_MTR_INST[i]._cfg.units = 4096.0 ;
						TML_MTR_INST[i]._cfg.rev_motor = 1;
						TML_MTR_INST[i]._cfg.rev_scale = 0.0375;  // this comes from experiment
						//TML_MTR_INST[i]._cfg.rev_scale = 1.0 / 56.0; // this comes from drawings
						TML_MTR_INST[i]._cfg.maxVel = 100.0;
						TML_MTR_INST[i]._cfg.maxAcc = 100.0;

						TML_MTR_INST[i]._cfg.AnalLimitPos = 3900;
						TML_MTR_INST[i]._cfg.AnalLimitNeg = 100;

					break;

					case TML_AX_TVL:

						strcpy(TML_MTR_INST[i].Name , "TVL");

						/// Deferent TML programs
						// Back EMF
						TML_MTR_INST[i]._cfg.loopPeriod = 0.001;

						if(ProjectConfig == project_US_Orbital){
							strcpy(TML_MTR_INST[i]._cfg.programName , "2511_TVL_D_HEAD_US.sw");
							TML_MTR_INST[i].ProgramVersion = ASC2UDINT("2511");
							TML_MTR_INST[i].FirmwareVersion = ASC2UDINT("6A2B");  //0x674B
							TML_MTR_INST[i]._cfg.Appl_ID_adr = 0x7FCF;

						}
						else{
							strcpy(TML_MTR_INST[i]._cfg.programName , "0411_TVL_FH_MINI_ENC.sw");
							TML_MTR_INST[i].ProgramVersion = ASC2UDINT("0411");
							TML_MTR_INST[i].FirmwareVersion = ASC2UDINT("674C");  //0x674C
						}

						TML_MTR_INST[i]._cfg.units =  1000; //  to jest tyle ile z max speed TML EREF
						//TML_MTR_INST[i]._cfg.rev_scale = -1920.0;
						TML_MTR_INST[i]._cfg.rev_scale =4000.0;
						TML_MTR_INST[i]._cfg.rev_motor = 1.0 ;
						TML_MTR_INST[i]._cfg.maxVel =  4; // mm/s
						TML_MTR_INST[i]._cfg.maxAcc = 100.0;
						TML_MTR_INST[i]._cfg.absFbk = 0; // non absolute value feedback , remember last value before drive reset

					break;

					default:

						xsprintf(TML_MTR_INST[i].Name, "Spare %d", i );
						TML_MTR_INST[i].pState = 0;

					break;

				}

			TML_MTR_INST[i].xCMD = TML_RESTART;

		}

		TML_mgr[0].hrdw[0].AxisNum = 3;
		TML_mgr[0].hrdw[1].AxisNum = 0;

		TML_mgr[0].pAxis[0] = &AxisCh[0];
		TML_mgr[0].pAxis[1] = 0;
		//TML_mgr[0].pAxis[1] = &AxisCh[TML_mgr[0].hrdw[0].AxisNum];

		TML_mgr[0].pTML[0] = &TML_MTR_INST[0];
		TML_mgr[0].pTML[1] = 0;
		//TML_mgr[0].pTML[1] = &TML_MTR_INST[TML_mgr[0].hrdw[0].AxisNum];

		AxisCh[TML_AX_TVL].AxisID	= 1;
		AxisCh[TML_AX_OSC].AxisID 	= 2;
		AxisCh[TML_AX_AVC].AxisID 	= 3;

		/**************************************/
		/****   Process   ************************/

		// Lincoln Power Supply
		for(i=0 ; i < 1; i++){

			switch(i){

				case 0:

					strcpy(Process[PROC_TIG_PS].Name , "TIG PS");
					PS_Param_Set[i].pPrc = &Process[PROC_TIG_PS];

					PS_Param_Set[i].pCalibPoints		= &m->pCalib->Points[CALIB_TIG_AMPS_CMD];
					//PS_Param_Set[i].rawCmdMax			= 26170; // //
					//PS_Param_Set[i].AmpCMD_Max			= 500.0; // 62.5 amp / 1 V
					PS_Param_Set[i].rawCmdMax			= 32767;
					PS_Param_Set[i].AmpCMD_Max			= 627.0;

					PS_Param_Set[i].pArcLinkRobot   = (UDINT)&ArcLink.robot;

				break;

			}

		}

		for(i=0 ; i < 1 ; i++){

			switch(i){

				case 0:

					strcpy(Process[PROC_AVC].Name , "AVC");

					strcpy(VectorStateMach[VECT_AVC].Name , "AVC");

					AVC_Param_Set[i].pPrc = &Process[PROC_AVC];
					AVC_Param_Set[i].pVect = &VectorStateMach[VECT_AVC];
					AVC_Param_Set[i].VectStateNum = 1;
					AVC_Param_Set[i].Mode = 0;

					AVC_Param_Set[i].MaxSpeedJog = 24.0;

					m->pCalib->Points[CALIB_TIG_VOLT_FBK].num = 10;
					AVC_Param_Set[i].pCalibPoints		= &m->pCalib->Points[CALIB_TIG_VOLT_FBK];

				break;

			}
		}

		for(i=0 ; i < 1 ; i++){

			switch(i){

				case 0:

					strcpy(Process[PROC_OSC].Name , "OSC");
					strcpy(VectorStateMach[VECT_OSC].Name , "OSC");

					OSC_TML_Param_Set[i].pPrc = &Process[PROC_OSC];
					OSC_TML_Param_Set[i].pVect = &VectorStateMach[VECT_OSC];
					OSC_TML_Param_Set[i].VectStateNum = 1;
					OSC_TML_Param_Set[i].pTML = &TML_MTR_INST[TML_AX_OSC] ;

					//OSC_TML_Param_Set[i].Mode = 0;
					OSC_TML_Param_Set[i].Mode = 11; // New Osc Mode -

					////  New Oscillation concept - BEMF
					OSC_TML_Param_Set[i].mm2ticks = TML_MTR_INST[TML_AX_OSC]._cfg.units * TML_MTR_INST[TML_AX_OSC]._cfg.rev_scale;
			 		OSC_TML_Param_Set[i].SpeedFactor = 410;
					//OSC_TML_Param_Set[i].MaxOscAmpl = 1.0 * 25.4;
					OSC_TML_Param_Set[i].MaxOscAmpl = 0.0;

					/////////////////////////
					/////   Hardcoded Limits
					if(cfg->HeadCfg.OSC.Limits_Harcoded){

						curCalib->Points[CALIB_OSC_SFT_LIMIT].num = 4;
						curCalib->Points[CALIB_OSC_SFT_LIMIT].val[0] = 10.0;
						curCalib->Points[CALIB_OSC_SFT_LIMIT].val[1] = 75.0;
						curCalib->Points[CALIB_OSC_SFT_LIMIT].val[2] = curCalib->Points[i].val[0];
						curCalib->Points[CALIB_OSC_SFT_LIMIT].val[3] = curCalib->Points[i].val[1];
					}

					////////////////////////////////////////////////

				break;

			}

		}

		for(i=0 ; i < 1 ; i++){

			switch(i){

				case 0:

					strcpy(Process[PROC_GAS].Name , "GAS");
					GAS_Param_Set[i].pPrc = &Process[PROC_GAS];

					//GAS_Param_Set[i].pSensInput     = &Hardware[1].Inp[5];  //FourAxis Head
					GAS_Param_Set[i].pOutput		= &Hardware[1].Outp[4];

				break;

			}

		}

		for(i=0 ; i < 1; i++){

			switch(i){

				case 0:

					strcpy(Process[PROC_COOL].Name , "COOLANT");
					COOL_Param_Set[i].pPrc = &Process[PROC_COOL];

					COOL_Param_Set[i].pSensInput     = &Hardware[1].Inp[4];  //FourAxis Head
					COOL_Param_Set[i].pOutput		= &Hardware[1].Outp[6];

				break;

			}

		}

		for(i=0 ; i < 1; i++){

			switch(i){

				case 0:

					strcpy(Process[PROC_HW_PS].Name , "HW PS");
					HW_PS_Param_Set[i].pPrc = &Process[PROC_HW_PS];

					HW_PS_Param_Set[i].pCalibPoints		= &m->pCalib->Points[CALIB_HW_AMPS_CMD];
					HW_PS_Param_Set[i].rawCmdMax 		= 16383.0;
					HW_PS_Param_Set[i].AmpCMD_Max 		= 160.0;

					Process[PROC_HW_PS].Disable = 1;

				break;

			}

		}

		for(i=0 ; i < 2; i++){

			switch(i){

				case 0:

					strcpy(Process[PROC_WIRE_FEED].Name ,"WrFeed");
					strcpy(VectorStateMach[VECT_WF].Name ,"WrFeed#1");
					strcpy(VectorStateMach[VECT_WF_1].Name ,"WrFeed#2");

					WIRE_Param_Set[i].pPrc = &Process[PROC_WIRE_FEED];
					WIRE_Param_Set[i].pVect = &VectorStateMach[m->pCfg->HeadCfg.WF.VECT_A_Indx];
					WIRE_Param_Set[i].VectStateNum = 1;
					WIRE_Param_Set[i].Mode = 0;  // classic

					WIRE_Param_Set[i].pCalibPoints	= &m->pCalib->Points[CALIB_WF_SPEED_CMD];

				break;

				case 1:

					strcpy(Process[PROC_WIRE_PULSE].Name ,"WrPulse");
					strcpy(VectorStateMach[VECT_WP].Name ,"WrPulse#1");
					strcpy(VectorStateMach[VECT_WP_1].Name ,"WrPulse#2");

					WIRE_Param_Set[i].pPrc = &Process[PROC_WIRE_PULSE];
					WIRE_Param_Set[i].pVect = &VectorStateMach[m->pCfg->HeadCfg.WP.VECT_A_Indx];
					WIRE_Param_Set[i].VectStateNum = 1;

					WIRE_Param_Set[i].pCalibPoints	= &m->pCalib->Points[CALIB_WP_SPEED_CMD];

					Process[PROC_WIRE_PULSE].Disable = 0;

				break;

		}

		}

		for(i=0 ; i < 1; i++){

			switch(i){

				case 0:

					strcpy(Process[PROC_TVL].Name , "TVL");
					strcpy(VectorStateMach[VECT_TVL].Name , "TVL");

					TVL_ROT_Param_Set[i].pPrc = &Process[PROC_TVL];
					TVL_ROT_Param_Set[i].pVect = &VectorStateMach[VECT_TVL];
					TVL_ROT_Param_Set[i].VectStateNum = 1;

					TVL_ROT_Param_Set[i].VectModeForJog = vectSt_Mode_Volt;

					TVL_ROT_Param_Set[i].MaxSpeedJog = 24.0;

					TVL_ROT_Param_Set[i].TotalRescaleFactor = 1.0;
					TVL_ROT_Param_Set[i].pCalibPoints = &m->pCalib->Points[CALIB_TVL_SPEED_CMD];

					TVL_ROT_Param_Set[i].pTrackDia = &curCfg->Param[parTVL_TrackDia].val[0];
					TVL_ROT_Param_Set[i].pVelTolerance = &curCfg->Param[parTVL_SpeedTolerane].val[0];

					TVL_ROT_Param_Set[i].pEncoder = &AxisCh[TML_AX_TVL].curPos;
					TVL_ROT_Param_Set[i].pHomePos = &OLD_MTR_POS[TVL_ENC_HOME];
					TVL_ROT_Param_Set[i].EncPerTick = m->pCfg->HeadCfg.TVL.EncPerTick;
					TVL_ROT_Param_Set[i].EncDir = m->pCfg->HeadCfg.TVL.Enc_Dir;
					TVL_ROT_Param_Set[i].TicksAtHighVel = 3;

				break;

			}
		}

		for(i=0 ; i < 1 ; i++){

			switch(i){

				case 0:

					strcpy(Process[m->pCfg->HeadCfg.INDX.PROC_Indx].Name , "INDX");
					INDEX_Param_Set[i].pPrc = &Process[m->pCfg->HeadCfg.INDX.PROC_Indx];
					Process[m->pCfg->HeadCfg.INDX.PROC_Indx].Disable = 1;

				break;

			}

		}

	return 1;

}

DINT Configure_U_BEND_HP_PINS(MASTER_typ * m,UINT headType){
return 1;
};

#if 0
DINT Configure_U_BEND_HP_PINS(MASTER_typ * m,UINT headType){
int i;

CurCfg_typ *curCfg;
Cfg_typ *cfg;
CurCalib_typ *curCalib , *defaultCalib;

	if(!m)
		return;

	curCfg = (CurCfg_typ*)m->pCurCfg;
	cfg = (Cfg_typ*)m->pCfg;

	curCalib = m->pCalib;
	defaultCalib = m->pDefaultCalib;

	if(!curCfg || !cfg || !curCalib  || !defaultCalib)
		return;

	/*********************************************/
	/***   Hardware and Vectors *********************/

	TML_MTR_INST[TML_AX_AVC].pState = &VectorStateMach[VECT_AVC];
	TML_MTR_INST[TML_AX_OSC].pState = &VectorStateMach[VECT_OSC];
	TML_MTR_INST[TML_AX_TVL].pState = &VectorStateMach[VECT_TVL];

	DC_Mtr[DC_AX_WF].pState = &VectorStateMach[VECT_WF];
	DC_Mtr[DC_AX_WP].pState = &VectorStateMach[VECT_WP];
	DC_Mtr[DC_AX_WF_1].pState = &VectorStateMach[VECT_WF_1];
	DC_Mtr[DC_AX_WP_1].pState = &VectorStateMach[VECT_WP_1];

#ifdef TEST_ONLY_PLC_ANDROID

	VectorStateMach[VECT_AVC].simul = 1;
	VectorStateMach[VECT_OSC].simul = 1;
	VectorStateMach[VECT_TVL].simul = 1;
	VectorStateMach[VECT_WF].simul = 1;
	VectorStateMach[VECT_WP].simul = 1;
	VectorStateMach[VECT_WF_1].simul = 1;
	VectorStateMach[VECT_WP_1].simul = 1;

	DC_Mtr[DC_AX_WF].Disable = 1;
	DC_Mtr[DC_AX_WP].Disable = 1;
	DC_Mtr[DC_AX_WF_1].Disable = 1;
	DC_Mtr[DC_AX_WP_1].Disable = 1;

	TML_MTR_INST[TML_AX_AVC].Disable = 1;
	TML_MTR_INST[TML_AX_OSC].Disable = 1;
	TML_MTR_INST[TML_AX_TVL].Disable = 1;

	//Process[PROC_AVC].Disable = 1;
	Process[PROC_AVC].TestMode = 1;
#endif

	/*********************************************************/
	/****   Phisical hardware configuration   ************************/

		for(i = 0 ; i < PROCESS_NUM; i++)
			strcpy(Process[i].Name , "spare");

		for(i = 0 ; i < VECTORS_NUM; i++)
			strcpy(VectorStateMach[i].Name , "spare");

		for(i = 0 ; i < GEN_MTR_NUM; i++){

			switch(i){

				case DC_AX_WF:
				case DC_AX_WF_1:

					switch(i){

						case DC_AX_WF:

							strcpy(DC_Mtr[i].Name , "DC WFeed#1");

							DC_Mtr[i].Cfg.mtr_dir = 1.0;
							DC_Mtr[i].Cfg.enc_dir = 1.0;

						break;

						case DC_AX_WF_1:

							strcpy(DC_Mtr[i].Name , "DC WFeed#2");

							DC_Mtr[i].Cfg.mtr_dir = 1.0;
							DC_Mtr[i].Cfg.enc_dir = 1.0;

						break;

					}

					//DC_Mtr[i].Cfg.units = 59.847340050885561192713356451475; // 0.75 " dia * 25.4 * PI
					DC_Mtr[i].Cfg.units = 2000 / 59.847340050885561192713356451475; // 2000 enc ticks / 0.75 " dia * 25.4 * PI
					DC_Mtr[i].Cfg.rev_scale = 66.0;	// Ratio gear box 66:1

					/* Parameters for PID controller */
					// To nowe
					DC_Mtr[i].msc.PIDParameters.Kp= 1.0;//0.4; //proportional gain / was 0.6
					//DC_Mtr[i].msc.PIDParameters.Kp= 0.1;//0.4; //proportional gain / was 0.6
					DC_Mtr[i].msc.PIDParameters.Tn= 0.1;//0.3.1; //intergral action time
					DC_Mtr[i].msc.PIDParameters.Kfbk = 0.01; //windup dampenin

					DC_Mtr[i].msc.PID.enable = 0;
					DC_Mtr[i].msc.PID.pPar = &DC_Mtr[i].msc.PIDParameters;
					DC_Mtr[i].msc.PID.request = 3; // Read parameters from PIDParameters
					DC_Mtr[i].msc.PIDParameters.Tv= 0; //derivative action time
					DC_Mtr[i].msc.PIDParameters.Y_max = 100.0;  //max manipulated variable %
					DC_Mtr[i].msc.PIDParameters.Y_min = -100.0; //min manipulated variable %

				break;

				case DC_AX_WP:
				case DC_AX_WP_1:

					switch(i){

						case DC_AX_WP:

							strcpy(DC_Mtr[i].Name , "DC WPulse#1");

							DC_Mtr[i].Cfg.mtr_dir = 1.0;
							DC_Mtr[i].Cfg.enc_dir = 1.0;

						break;

						case DC_AX_WP_1:

							strcpy(DC_Mtr[i].Name , "DC WPulse#2");

							DC_Mtr[i].Cfg.mtr_dir = 1.0;
							DC_Mtr[i].Cfg.enc_dir = 1.0;

						break;

					}

					//oryginalnie jest 2000 pulsow na obrot potem ratio on gear 4.8 : 1
					DC_Mtr[i].Cfg.units = 2000;
					DC_Mtr[i].Cfg.rev_scale = 4.8;// ratio on gear 4.8

					/* Parameters for PID controller */
					// To nowe
					DC_Mtr[i].msc.PIDParameters.Kp= 1.0;//0.4; //proportional gain / was 0.6
					//DC_Mtr[i].msc.PIDParameters.Kp= 0.1;//0.4; //proportional gain / was 0.6
					DC_Mtr[i].msc.PIDParameters.Tn= 0.1;//0.3.1; //intergral action time
					DC_Mtr[i].msc.PIDParameters.Kfbk = 0.01; //windup dampenin

					DC_Mtr[i].msc.PID.enable = 0;
					DC_Mtr[i].msc.PID.pPar = &DC_Mtr[i].msc.PIDParameters;
					DC_Mtr[i].msc.PID.request = 3; // Read parameters from PIDParameters
					DC_Mtr[i].msc.PIDParameters.Tv= 0; //derivative action time
					DC_Mtr[i].msc.PIDParameters.Y_max = 100.0;  //max manipulated variable %
					DC_Mtr[i].msc.PIDParameters.Y_min = -100.0; //min manipulated variable %

				break;

				default:

					strcpy(DC_Mtr[i].Name , "Spare ");

				break;

			}

			//CalcUnits(&DC_Mtr[i]);
			DC_Mtr[i].msc.kPos = (float)DC_Mtr[i].Cfg.units * DC_Mtr[i].Cfg.rev_scale;

		}

		/***********************************/

			for(i = 0 ; i < TML_SERVO_NUM ; i++){

				switch(i){

					// tml->_int.kPos = (tml->_cfg.units * tml->_cfg.rev_scale) / tml->_cfg.rev_motor;
					case TML_AX_AVC:

						strcpy(TML_MTR_INST[i].Name , "AVC");

						// Analog Feedback from REF
						TML_MTR_INST[i]._cfg.loopPeriod = 0.001;
						TML_MTR_INST[i]._cfg.units = 4095;
						TML_MTR_INST[i]._cfg.rev_motor = 1;
						TML_MTR_INST[i]._cfg.rev_scale = 1.0/5.0;
						TML_MTR_INST[i]._cfg.maxVel = 1.0; //1//6000 rpm
						TML_MTR_INST[i]._cfg.maxAcc = 100.0;
						//TML_MTR_INST[i]._cfg.satpMax = 27853; // KPP bylo Stauration of proportional gain
						TML_MTR_INST[i]._cfg.satpMax = 32000; // KPP bylo Stauration of proportional gain
						TML_MTR_INST[i]._cfg.kppMax = 32000; // KPP bylo Stauration of proportional gain
						TML_MTR_INST[i]._cfg.kipMax = 200; // KPP bylo Stauration of proportional gain
						TML_MTR_INST[i]._cfg.absFbk = 0; // absolute value feedback

						TML_MTR_INST[i]._cfg.signFilter = curCfg->Param[parAVC_FbkFilter].val[0];

						//U_BEND_HP_PINS
						strcpy(TML_MTR_INST[i]._cfg.programName , "0013_AVC_U_BEND_HP_PINS.sw");
						TML_MTR_INST[i].ProgramVersion = ASC2UDINT("0013");

						TML_MTR_INST[i].FirmwareVersion = ASC2UDINT("674C");  //0x674C

						//TML_MTR_INST[i]._cfg.sftLimitPos = 1000.0;
						//TML_MTR_INST[i]._cfg.sftLimitNeg = -1000.0;

					break;

					case TML_AX_OSC:

						strcpy(TML_MTR_INST[i].Name , "OSC");

						// Analog Feedback from REF
						TML_MTR_INST[i]._cfg.loopPeriod = 0.001;

						TML_MTR_INST[i]._cfg.units = 80;
						TML_MTR_INST[i]._cfg.rev_motor = 1;
						TML_MTR_INST[i]._cfg.rev_scale = 1.0;
						TML_MTR_INST[i]._cfg.maxVel = 100.0; //1//6000 rpm
						TML_MTR_INST[i]._cfg.maxAcc = 100.0;
						TML_MTR_INST[i]._cfg.absFbk = 0; // absolute value feedback

						// U_BEND_HP_PINS
						strcpy(TML_MTR_INST[i]._cfg.programName , "0012_OSC_U_BEND_HP_PINS.sw");
						TML_MTR_INST[i].ProgramVersion = ASC2UDINT("0012");

						TML_MTR_INST[i].FirmwareVersion = ASC2UDINT("674C");  //0x674B

						//TML_MTR_INST[i]._cfg.sftLimitPos = curCalib->Points[CALIB_OSC_SFT_LIMIT].val[0];

						//TML_MTR_INST[i]._cfg.sftLimitNeg = curCalib->Points[CALIB_OSC_SFT_LIMIT].val[1];

					break;

					case TML_AX_TVL:

						strcpy(TML_MTR_INST[i].Name , "TVL");
						// Back EMF
						TML_MTR_INST[i]._cfg.loopPeriod = 0.001;
						TML_MTR_INST[i]._cfg.units = 1000 * 60; // unit rps/sec
						TML_MTR_INST[i]._cfg.rev_motor = 1;
						TML_MTR_INST[i]._cfg.rev_scale = 10.2;
						TML_MTR_INST[i]._cfg.maxVel =  3.0; // mm/s
						TML_MTR_INST[i]._cfg.maxAcc = 20.0;
						TML_MTR_INST[i]._cfg.absFbk = 0; // non absolute value feedback , remember last value before drive reset

						//* U_BEND_HP_PINS
						strcpy(TML_MTR_INST[i]._cfg.programName , "0011_TVL_U_BEND_HP_PINS.sw");
						TML_MTR_INST[i].ProgramVersion = ASC2UDINT("0011");

						TML_MTR_INST[i].FirmwareVersion = ASC2UDINT("674C");  //0x674B

					break;

					default:

						xsprintf(TML_MTR_INST[i].Name, "Spare %d", i );
						TML_MTR_INST[i].pState = 0;

					break;

				}

			TML_MTR_INST[i].xCMD = TML_RESTART;

		}

		TML_mgr[0].hrdw[0].AxisNum = 3;
		TML_mgr[0].hrdw[1].AxisNum = 0;

		TML_mgr[0].pAxis[0] = &AxisCh[0];
		TML_mgr[0].pAxis[1] = 0;
		//TML_mgr[0].pAxis[1] = &AxisCh[TML_mgr[0].hrdw[0].AxisNum];

		TML_mgr[0].pTML[0] = &TML_MTR_INST[0];
		TML_mgr[0].pTML[1] = 0;
		//TML_mgr[0].pTML[1] = &TML_MTR_INST[TML_mgr[0].hrdw[0].AxisNum];

		AxisCh[TML_AX_TVL].AxisID	= 1;
		AxisCh[TML_AX_OSC].AxisID 	= 2;
		AxisCh[TML_AX_AVC].AxisID 	= 3;

		/**************************************/
		/****   Process   ************************/

		for(i=0 ; i < 1; i++){

			switch(i){

				case 0:

					strcpy(Process[PROC_TIG_PS].Name , "TIG PS");
					PS_Param_Set[i].pPrc = &Process[PROC_TIG_PS];

					/*
					// This is only when we use two analog aoutputs to reach 15V
					PS_Param_Set[i].pCalibPoints		= &m->pCalib->Points[CALIB_TIG_AMPS_CMD];
					PS_Param_Set[i].rawCmdMax			= 26170; // //
					PS_Param_Set[i].AmpCMD_Max			= 500.0; // 62.5 amp / 1 V
					*/

					// Only one analog output - 10V -> 345 Amps
					PS_Param_Set[i].pCalibPoints		= &m->pCalib->Points[CALIB_TIG_AMPS_CMD];
					PS_Param_Set[i].rawCmdMax 			= 32767.0;
					//PS_Param_Set[i].AmpCMD_Max		= 345.0;
					PS_Param_Set[i].AmpCMD_Max			= 500.0; // new firmware

				break;

			}

		}

		for(i=0 ; i < 1 ; i++){

			switch(i){

				case 0:

					strcpy(Process[PROC_AVC].Name , "AVC");

					strcpy(VectorStateMach[VECT_AVC].Name , "AVC");

					AVC_Param_Set[i].pPrc = &Process[PROC_AVC];
					AVC_Param_Set[i].pVect = &VectorStateMach[VECT_AVC];
					AVC_Param_Set[i].VectStateNum = 1;

					m->pCalib->Points[CALIB_TIG_VOLT_FBK].num = 10;
					AVC_Param_Set[i].pCalibPoints		= &m->pCalib->Points[CALIB_TIG_VOLT_FBK];

				break;

			}
		}

		for(i=0 ; i < 1 ; i++){

			switch(i){

				case 0:

					strcpy(Process[PROC_OSC].Name , "OSC");
					strcpy(VectorStateMach[VECT_OSC].Name , "OSC");

					OSC_TML_Param_Set[i].pPrc = &Process[PROC_OSC];
					OSC_TML_Param_Set[i].pVect = &VectorStateMach[VECT_OSC];
					OSC_TML_Param_Set[i].VectStateNum = 1;
					OSC_TML_Param_Set[i].pTML = &TML_MTR_INST[TML_AX_OSC] ;

				break;

			}

		}

		for(i=0 ; i < 1 ; i++){

			switch(i){

				case 0:

					strcpy(Process[PROC_GAS].Name , "GAS");
					GAS_Param_Set[i].pPrc = &Process[PROC_GAS];

					//GAS_Param_Set[i].pSensInput     = &Hardware[1].Inp[5];  //FourAxis Head
					GAS_Param_Set[i].pOutput		= &Hardware[1].Outp[4];

				break;

			}

		}

		for(i=0 ; i < 1; i++){

			switch(i){

				case 0:

					strcpy(Process[PROC_COOL].Name , "COOLANT");
					COOL_Param_Set[i].pPrc = &Process[PROC_COOL];

					COOL_Param_Set[i].pSensInput     = &Hardware[1].Inp[4];  //FourAxis Head
					COOL_Param_Set[i].pOutput		= &Hardware[1].Outp[6];

				break;

			}

		}

		for(i=0 ; i < 1; i++){

			switch(i){

				case 0:

					strcpy(Process[PROC_HW_PS].Name , "HW PS");
					HW_PS_Param_Set[i].pPrc = &Process[PROC_HW_PS];

					HW_PS_Param_Set[i].pCalibPoints		= &m->pCalib->Points[CALIB_HW_AMPS_CMD];
					HW_PS_Param_Set[i].rawCmdMax 		= 16383.0;
					HW_PS_Param_Set[i].AmpCMD_Max 		= 160.0;

				break;

			}

		}

		for(i=0 ; i < 2; i++){

			switch(i){

				case 0:

					strcpy(Process[PROC_WIRE_FEED].Name ,"WrFeed");
					strcpy(VectorStateMach[VECT_WF].Name ,"WrFeed#1");
					strcpy(VectorStateMach[VECT_WF_1].Name ,"WrFeed#2");

					WIRE_Param_Set[i].pPrc = &Process[PROC_WIRE_FEED];
					WIRE_Param_Set[i].pVect = &VectorStateMach[VECT_WF];
					WIRE_Param_Set[i].VectStateNum = 1;

					WIRE_Param_Set[i].pCalibPoints	= &m->pCalib->Points[CALIB_WF_SPEED_CMD];

				break;

				case 1:

					strcpy(Process[PROC_WIRE_PULSE].Name ,"WrPulse");
					strcpy(VectorStateMach[VECT_WP].Name ,"WrPulse#1");
					strcpy(VectorStateMach[VECT_WP_1].Name ,"WrPulse#2");

					WIRE_Param_Set[i].pPrc = &Process[PROC_WIRE_PULSE];
					WIRE_Param_Set[i].pVect = &VectorStateMach[VECT_WP];
					WIRE_Param_Set[i].VectStateNum = 1;

					WIRE_Param_Set[i].pCalibPoints	= &m->pCalib->Points[CALIB_WP_SPEED_CMD];

				break;

		}

		}

		for(i=0 ; i < 1; i++){

			switch(i){

				case 0:

					strcpy(Process[PROC_TVL].Name , "TVL");
					strcpy(VectorStateMach[VECT_TVL].Name , "TVL");

					TVL_ROT_Param_Set[i].pPrc = &Process[PROC_TVL];
					TVL_ROT_Param_Set[i].pVect = &VectorStateMach[VECT_TVL];
					TVL_ROT_Param_Set[i].VectStateNum = 1;

					TVL_ROT_Param_Set[i].VectModeForJog = vectSt_Mode_Volt;

					TVL_ROT_Param_Set[i].TotalRescaleFactor = 1.0;
					TVL_ROT_Param_Set[i].pCalibPoints = &m->pCalib->Points[CALIB_TVL_SPEED_CMD];

					TVL_ROT_Param_Set[i].pTrackDia = &curCfg->Param[parTVL_TrackDia].val[0];
					TVL_ROT_Param_Set[i].pVelTolerance = &curCfg->Param[parTVL_SpeedTolerane].val[0];

				break;

			}

		}

		for(i=0 ; i < 1 ; i++){

			switch(i){

				case 0:

					strcpy(Process[m->pCfg->HeadCfg.INDX.PROC_Indx].Name , "INDX");
					INDEX_Param_Set[i].pPrc = &Process[m->pCfg->HeadCfg.INDX.PROC_Indx];
					Process[m->pCfg->HeadCfg.INDX.PROC_Indx].Disable = 1;

				break;

			}

		}

	// One oscillator
	//m->OscNum = 1;

	//m->directTVL = -1;

	return 1;

}
#endif

DINT Configure_U_BEND_HP_ENC(MASTER_typ * m,UINT headType){
int i;

CurCfg_typ *curCfg;
Cfg_typ *cfg;
CurCalib_typ *curCalib , *defaultCalib;

	if(!m)
		return;

	curCfg = (CurCfg_typ*)m->pCurCfg;
	cfg = (Cfg_typ*)m->pCfg;

	curCalib = m->pCalib;
	defaultCalib = m->pDefaultCalib;

	if(!curCfg || !cfg || !curCalib  || !defaultCalib)
		return;

	/*********************************************/
	/***   Hardware and Vectors *********************/

	TML_MTR_INST[m->pCfg->HeadCfg.TVL.TML_Indx ].pState = &VectorStateMach[m->pCfg->HeadCfg.TVL.VECT_Indx];

	TML_MTR_INST[m->pCfg->HeadCfg.AVC.TML_A_Indx ].pState = &VectorStateMach[m->pCfg->HeadCfg.AVC.VECT_A_Indx];
	TML_MTR_INST[m->pCfg->HeadCfg.AVC.TML_B_Indx ].pState = &VectorStateMach[m->pCfg->HeadCfg.AVC.VECT_B_Indx];

	TML_MTR_INST[m->pCfg->HeadCfg.OSC.TML_A_Indx ].pState = &VectorStateMach[m->pCfg->HeadCfg.OSC.VECT_A_Indx];
	TML_MTR_INST[m->pCfg->HeadCfg.OSC.TML_B_Indx ].pState = &VectorStateMach[m->pCfg->HeadCfg.OSC.VECT_B_Indx];

	DC_Mtr[m->pCfg->HeadCfg.WF.DC_A_Indx ].pState = &VectorStateMach[m->pCfg->HeadCfg.WF.VECT_A_Indx];
	DC_Mtr[m->pCfg->HeadCfg.WP.DC_A_Indx ].pState = &VectorStateMach[m->pCfg->HeadCfg.WP.VECT_A_Indx];
	DC_Mtr[m->pCfg->HeadCfg.WF.DC_B_Indx ].pState = &VectorStateMach[m->pCfg->HeadCfg.WF.VECT_B_Indx];
	DC_Mtr[m->pCfg->HeadCfg.WP.DC_B_Indx ].pState = &VectorStateMach[m->pCfg->HeadCfg.WP.VECT_B_Indx];

#ifdef SYSTEM_SIMULATION

	VectorStateMach[VECT_AVC].simul = 1;
	VectorStateMach[VECT_OSC].simul = 1;
	VectorStateMach[VECT_TVL].simul = 1;
	VectorStateMach[VECT_WF].simul = 1;
	VectorStateMach[VECT_WP].simul = 1;
	VectorStateMach[VECT_WF_1].simul = 1;
	VectorStateMach[VECT_WP_1].simul = 1;

	DC_Mtr[DC_AX_WF].Disable = 1;
	DC_Mtr[DC_AX_WP].Disable = 1;
	DC_Mtr[DC_AX_WF_1].Disable = 1;
	DC_Mtr[DC_AX_WP_1].Disable = 1;

	TML_MTR_INST[TML_AX_AVC].Disable = 1;
	TML_MTR_INST[TML_AX_OSC].Disable = 1;
	TML_MTR_INST[TML_AX_TVL].Disable = 1;

	//Process[PROC_AVC].Disable = 1;
	Process[PROC_AVC].TestMode = 1;

#else

	Process[PROC_TVL].Disable = 0;
	Process[PROC_OSC].Disable = 0;
	Process[PROC_AVC].Disable = 0;
	Process[PROC_WIRE_FEED].Disable = 0;
	Process[PROC_WIRE_PULSE].Disable = 0;

	VectorStateMach[VECT_AVC].simul = 0;
	VectorStateMach[VECT_OSC].simul = 0;
	VectorStateMach[VECT_TVL].simul = 0;

	VectorStateMach[VECT_WF].simul 		= 0;
	VectorStateMach[VECT_WF_1].simul 	= 0;
	VectorStateMach[VECT_WP].simul 		= 0;
	VectorStateMach[VECT_WP_1].simul 	= 0;

	DC_Mtr[DC_AX_WF].Disable = 0;
	DC_Mtr[DC_AX_WP].Disable = 0;
	DC_Mtr[DC_AX_WF_1].Disable = 0;
	DC_Mtr[DC_AX_WP_1].Disable = 0;

	TML_MTR_INST[TML_AX_AVC].Disable = 0;
	TML_MTR_INST[TML_AX_OSC].Disable = 0;
	TML_MTR_INST[TML_AX_TVL].Disable = 0;

#endif

	/*********************************************************/
	/****   Phisical hardware configuration   ************************/

		for(i = 0 ; i < PROCESS_NUM; i++)
			strcpy(Process[i].Name , "spare");

		for(i = 0 ; i < VECTORS_NUM; i++)
			strcpy(VectorStateMach[i].Name , "spare");

		//////////////////////////////////////////////////////////////////////////////////
		// Wire Block
		for(i=0 ; i < 2; i++){

			switch(i){

				case 0:
					strcpy(Process[m->pCfg->HeadCfg.WB[i].PROC_Indx].Name , "WB_UD");
					strcpy(VectorStateMach[m->pCfg->HeadCfg.WB[i].VECT_Indx].Name , "WB_UD");

					WR_BLK_Param_Set[i].pPrc = &Process[m->pCfg->HeadCfg.WB[i].PROC_Indx];
					WR_BLK_Param_Set[i].pVect = &VectorStateMach[m->pCfg->HeadCfg.WB[i].VECT_Indx];
					WR_BLK_Param_Set[i].VectStateNum = 1;

					WR_BLK_Param_Set[i].MaxSpeedJog = 24.0;

					Gen_one = 1.0;
					WR_BLK_Param_Set[i].pJogSpeed = &Gen_one;

				break;

				case 1:
					strcpy(Process[m->pCfg->HeadCfg.WB[i].PROC_Indx].Name , "WB_LR");
					strcpy(VectorStateMach[m->pCfg->HeadCfg.WB[i].VECT_Indx].Name , "WB_LR");

					WR_BLK_Param_Set[i].pPrc = &Process[PROC_WB_LR];
					WR_BLK_Param_Set[i].pVect = &VectorStateMach[VECT_WB_LR];
					WR_BLK_Param_Set[i].VectStateNum = 1;

					WR_BLK_Param_Set[i].MaxSpeedJog = 24.0;

					Gen_one = 1.0;
					WR_BLK_Param_Set[i].pJogSpeed = &Gen_one;

				break;

			}

		}

		for(i = 0 ; i < DC2DIRMTR_NUM; i++){

			switch(i){

				case DC_WB_UD:

					strcpy(DC2DirMtr[i].Name , "WB_UD");
					DC2DirMtr[i].pState = &VectorStateMach[VECT_WB_UD];

					DC2DirMtr[i].Cfg.pQ1_output = &Hardware[1].Outp[12];
					DC2DirMtr[i].Cfg.pQ2_output = &Hardware[1].Outp[13];
					DC2DirMtr[i].Cfg.pQ3_output = &Hardware[1].Outp[14];
					DC2DirMtr[i].Cfg.pQ4_output = &Hardware[1].Outp[15];

					DC2DirMtr[i].Cfg.MtrDir = 1.0;

				break;

				case DC_WB_LR:

					strcpy(DC2DirMtr[i].Name , "WB_LR");
					DC2DirMtr[i].pState = &VectorStateMach[VECT_WB_LR];

					DC2DirMtr[i].Cfg.pQ1_output = &Hardware[1].Outp[16];
					DC2DirMtr[i].Cfg.pQ2_output = &Hardware[1].Outp[17];
					DC2DirMtr[i].Cfg.pQ3_output = &Hardware[1].Outp[18];
					DC2DirMtr[i].Cfg.pQ4_output = &Hardware[1].Outp[19];

					DC2DirMtr[i].Cfg.MtrDir = 1.0;

				break;

			}

		}
		/////////////////////////////////////////////////////////////////////////////////

		for(i = 0 ; i < GEN_MTR_NUM; i++){

			switch(i){

				case DC_AX_WF:
				case DC_AX_WF_1:

					switch(i){

						case DC_AX_WF:

							strcpy(DC_Mtr[i].Name , "DC WFeed#1");

							DC_Mtr[i].Cfg.mtr_dir = -1.0;

							if(ProjectConfig == project_US_Orbital) // US Orbital has B and /B swapped
								DC_Mtr[i].Cfg.enc_dir = -1.0;
							else
								DC_Mtr[i].Cfg.enc_dir = 1.0;

						break;

						case DC_AX_WF_1:

							strcpy(DC_Mtr[i].Name , "DC WFeed#2");

							DC_Mtr[i].Cfg.mtr_dir = 1.0;

							if(ProjectConfig == project_US_Orbital) // US Orbital has B and /B swapped
								DC_Mtr[i].Cfg.enc_dir = -1.0;
							else
								DC_Mtr[i].Cfg.enc_dir = 1.0;

						break;

					}

					//DC_Mtr[i].Cfg.units = 59.847340050885561192713356451475; // 0.75 " dia * 25.4 * PI
					DC_Mtr[i].Cfg.units = 2000 / 59.847340050885561192713356451475; // 2000 enc ticks / 0.75 " dia * 25.4 * PI
					DC_Mtr[i].Cfg.rev_scale = 66.0;	// Ratio gear box 66:1

					/* Parameters for PID controller */
					// To nowe
					DC_Mtr[i].msc.PIDParameters.Kp= 1.0;//0.4; //proportional gain / was 0.6
					//DC_Mtr[i].msc.PIDParameters.Kp= 0.1;//0.4; //proportional gain / was 0.6
					DC_Mtr[i].msc.PIDParameters.Tn= 0.1;//0.3.1; //intergral action time
					DC_Mtr[i].msc.PIDParameters.Kfbk = 0.01; //windup dampenin

					DC_Mtr[i].msc.PID.enable = 0;
					DC_Mtr[i].msc.PID.pPar = &DC_Mtr[i].msc.PIDParameters;
					DC_Mtr[i].msc.PID.request = 3; // Read parameters from PIDParameters
					DC_Mtr[i].msc.PIDParameters.Tv= 0; //derivative action time
					DC_Mtr[i].msc.PIDParameters.Y_max = 100.0;  //max manipulated variable %
					DC_Mtr[i].msc.PIDParameters.Y_min = -100.0; //min manipulated variable %

				break;

				case DC_AX_WP:
				case DC_AX_WP_1:

					switch(i){

						case DC_AX_WP:

							strcpy(DC_Mtr[i].Name , "DC WPulse#1");

							DC_Mtr[i].Cfg.mtr_dir = 1.0;

							if(ProjectConfig == project_US_Orbital) // US Orbital has B and /B swapped
								DC_Mtr[i].Cfg.enc_dir = -1.0;
							else
								DC_Mtr[i].Cfg.enc_dir = 1.0;

						break;

						case DC_AX_WP_1:

							strcpy(DC_Mtr[i].Name , "DC WPulse#2");

							DC_Mtr[i].Cfg.mtr_dir = 1.0;

							if(ProjectConfig == project_US_Orbital) // US Orbital has B and /B swapped
								DC_Mtr[i].Cfg.enc_dir = -1.0;
							else
								DC_Mtr[i].Cfg.enc_dir = 1.0;

						break;

					}

					//oryginalnie jest 2000 pulsow na obrot potem ratio on gear 4.8 : 1
					DC_Mtr[i].Cfg.units = 2000;
					DC_Mtr[i].Cfg.rev_scale = 4.8;// ratio on gear 4.8

					/* Parameters for PID controller */
					// To nowe
					DC_Mtr[i].msc.PIDParameters.Kp= 1.0;//0.4; //proportional gain / was 0.6
					//DC_Mtr[i].msc.PIDParameters.Kp= 0.1;//0.4; //proportional gain / was 0.6
					DC_Mtr[i].msc.PIDParameters.Tn= 0.1;//0.3.1; //intergral action time
					DC_Mtr[i].msc.PIDParameters.Kfbk = 0.01; //windup dampenin

					DC_Mtr[i].msc.PID.enable = 0;
					DC_Mtr[i].msc.PID.pPar = &DC_Mtr[i].msc.PIDParameters;
					DC_Mtr[i].msc.PID.request = 3; // Read parameters from PIDParameters
					DC_Mtr[i].msc.PIDParameters.Tv= 0; //derivative action time
					DC_Mtr[i].msc.PIDParameters.Y_max = 100.0;  //max manipulated variable %
					DC_Mtr[i].msc.PIDParameters.Y_min = -100.0; //min manipulated variable %

				break;

				default:

					//strcpy(DC_Mtr[i].Name , "Spare ");
					xsprintf(DC_Mtr[i].Name, "Spare %d", i );

				break;

			}

			//CalcUnits(&DC_Mtr[i]);
			DC_Mtr[i].msc.kPos = (float)DC_Mtr[i].Cfg.units * DC_Mtr[i].Cfg.rev_scale;

		}

		/***********************************/

			for(i = 0 ; i < TML_SERVO_NUM ; i++){

				switch(i){

					// tml->_int.kPos = (tml->_cfg.units * tml->_cfg.rev_scale) / tml->_cfg.rev_motor;
					case TML_AX_AVC:

						strcpy(TML_MTR_INST[i].Name , "AVC");

						// Analog Feedback from REF
						TML_MTR_INST[i]._cfg.loopPeriod = 0.001;
						TML_MTR_INST[i]._cfg.units = 4095;
						//TML_MTR_INST[i]._cfg.rev_motor = 1;
						TML_MTR_INST[i]._cfg.rev_scale = 1.0/5.0;
						TML_MTR_INST[i]._cfg.maxVel = 10.0; //1//6000 rpm
						TML_MTR_INST[i]._cfg.maxAcc = 100000.0;
						//TML_MTR_INST[i]._cfg.satpMax = 27853; // KPP bylo Stauration of proportional gain
						TML_MTR_INST[i]._cfg.satpMax = 32000; // KPP bylo Stauration of proportional gain
						//TML_MTR_INST[i]._cfg.kppMax = 32000; // KPP bylo Stauration of proportional gain
						//TML_MTR_INST[i]._cfg.kipMax = 200; // KPP bylo Stauration of proportional gain
						TML_MTR_INST[i]._cfg.absFbk = 0; // absolute value feedback

						TML_MTR_INST[i]._cfg.signFilter = curCfg->Param[parAVC_FbkFilter].val[0];

						if(ProjectConfig == project_US_Orbital){
							strcpy(TML_MTR_INST[i]._cfg.programName , "1023_AVC_U_BEND_ENC_US.sw");
							TML_MTR_INST[i].ProgramVersion = ASC2UDINT("1023");
							TML_MTR_INST[i].FirmwareVersion = ASC2UDINT("6A2B");  //0x674B
							TML_MTR_INST[i]._cfg.Appl_ID_adr = 0x7FCF;
							TML_MTR_INST[i]._cfg.rev_motor = -1.0;
							TML_MTR_INST[i]._cfg.kppMax = -32000; // KPP bylo Stauration of proportional gain
							TML_MTR_INST[i]._cfg.kipMax = -200; // KPP bylo Stauration of proportional gain

						}
						else{
							strcpy(TML_MTR_INST[i]._cfg.programName , "0023_AVC_U_BEND_ENC.sw");
							TML_MTR_INST[i].ProgramVersion = ASC2UDINT("0023");
							TML_MTR_INST[i].FirmwareVersion = ASC2UDINT("674C");  //0x674C
							TML_MTR_INST[i]._cfg.rev_motor = 1.0;
							TML_MTR_INST[i]._cfg.kppMax = 32000; // KPP bylo Stauration of proportional gain
							TML_MTR_INST[i]._cfg.kipMax = 200; // KPP bylo Stauration of proportional gain
						}

						//TML_MTR_INST[i]._cfg.sftLimitPos = 1000.0;
						//TML_MTR_INST[i]._cfg.sftLimitNeg = -1000.0;

					break;

					case TML_AX_OSC:

						strcpy(TML_MTR_INST[i].Name , "OSC");

						if(ProjectConfig == project_US_Orbital){
							strcpy(TML_MTR_INST[i]._cfg.programName , "1022_OSC_U_BEND_ENC_US.sw");
							TML_MTR_INST[i].ProgramVersion = ASC2UDINT("1022");
							TML_MTR_INST[i].FirmwareVersion = ASC2UDINT("6A2B");  //0x674B
							TML_MTR_INST[i]._cfg.Appl_ID_adr = 0x7FCF;
							TML_MTR_INST[i]._cfg.rev_motor = -1.0;

						}
						else{
							strcpy(TML_MTR_INST[i]._cfg.programName , "0022_OSC_U_BEND_ENC.sw");
							TML_MTR_INST[i].ProgramVersion = ASC2UDINT("0022");
							TML_MTR_INST[i].FirmwareVersion = ASC2UDINT("674C");  //0x674C
							TML_MTR_INST[i]._cfg.rev_motor = 1.0;

						}

						TML_MTR_INST[i]._cfg.loopPeriod = 0.001;
						TML_MTR_INST[i]._cfg.absFbk = 0; // value fom APOS which is analog Ref
						TML_MTR_INST[i]._cfg.units = 4096.0 ;
						//TML_MTR_INST[i]._cfg.rev_motor = 1;
						TML_MTR_INST[i]._cfg.rev_scale = 1.0 / 80.0;  // this comes from experiment
						//TML_MTR_INST[i]._cfg.rev_scale = 1.0 / 56.0; // this comes from drawings
						TML_MTR_INST[i]._cfg.maxVel = 100.0;
						TML_MTR_INST[i]._cfg.maxAcc = 100.0;

						TML_MTR_INST[i]._cfg.AnalLimitPos = 3900;
						TML_MTR_INST[i]._cfg.AnalLimitNeg = 100;

					break;

					case TML_AX_TVL:

						strcpy(TML_MTR_INST[i].Name , "TVL");

						/// Deferent TML programs
						// Back EMF
						TML_MTR_INST[i]._cfg.loopPeriod = 0.001;

						if(ProjectConfig == project_US_Orbital){
							strcpy(TML_MTR_INST[i]._cfg.programName , "1021_TVL_U_BEND_ENC_US.sw");
							TML_MTR_INST[i].ProgramVersion = ASC2UDINT("1021");
							TML_MTR_INST[i].FirmwareVersion = ASC2UDINT("6A2B");  //0x674B
							TML_MTR_INST[i]._cfg.Appl_ID_adr = 0x7FCF;
							TML_MTR_INST[i]._cfg.rev_motor = -1.0;
							TML_MTR_INST[i]._cfg.rev_scale = -1920.0;

						}
						else{
							strcpy(TML_MTR_INST[i]._cfg.programName , "0021_TVL_U_BEND_ENC.sw");
							TML_MTR_INST[i].ProgramVersion = ASC2UDINT("0021");
							TML_MTR_INST[i].FirmwareVersion = ASC2UDINT("674C");  //0x674C
							TML_MTR_INST[i]._cfg.rev_motor = -1.0;
							TML_MTR_INST[i]._cfg.rev_scale = -1920.0;
						}

						TML_MTR_INST[i]._cfg.units =  1000; //  to jest tyle ile z max speed TML EREF
						//TML_MTR_INST[i]._cfg.rev_scale = -1920.0;
						//TML_MTR_INST[i]._cfg.rev_motor = 1.0 ;
						TML_MTR_INST[i]._cfg.maxVel =  10.0; // mm/s
						TML_MTR_INST[i]._cfg.maxAcc = 100.0;
						TML_MTR_INST[i]._cfg.absFbk = 0; // non absolute value feedback , remember last value before drive reset

					break;

					default:

						//xsprintf(TML_MTR_INST[i].Name, "Spare %d", i );
						xsprintf(TML_MTR_INST[i].Name, "Spare %d", i );

					break;

				}

			TML_MTR_INST[i].xCMD = TML_RESTART;

		}

		TML_mgr[0].hrdw[0].AxisNum = 3;
		TML_mgr[0].hrdw[1].AxisNum = 0;

		TML_mgr[0].pAxis[0] = &AxisCh[0];
		TML_mgr[0].pAxis[1] = 0;
		//TML_mgr[0].pAxis[1] = &AxisCh[TML_mgr[0].hrdw[0].AxisNum];

		TML_mgr[0].pTML[0] = &TML_MTR_INST[0];
		TML_mgr[0].pTML[1] = 0;
		//TML_mgr[0].pTML[1] = &TML_MTR_INST[TML_mgr[0].hrdw[0].AxisNum];

		AxisCh[TML_AX_TVL].AxisID	= 1;
		AxisCh[TML_AX_OSC].AxisID 	= 2;
		AxisCh[TML_AX_AVC].AxisID 	= 3;

		/**************************************/
		/****   Process   ************************/

		// Lincoln Power Supply
		for(i=0 ; i < 1; i++){

			switch(i){

				case 0:

					strcpy(Process[PROC_TIG_PS].Name , "TIG PS");
					PS_Param_Set[i].pPrc = &Process[PROC_TIG_PS];

					PS_Param_Set[i].pCalibPoints		= &m->pCalib->Points[CALIB_TIG_AMPS_CMD];
					//PS_Param_Set[i].rawCmdMax			= 26170; // //
					//PS_Param_Set[i].AmpCMD_Max			= 500.0; // 62.5 amp / 1 V
					PS_Param_Set[i].rawCmdMax			= 32767;
					PS_Param_Set[i].AmpCMD_Max			= 627.0;

					PS_Param_Set[i].pArcLinkRobot   = (UDINT)&ArcLink.robot;

				break;

			}

		}

		for(i=0 ; i < 1 ; i++){

			switch(i){

				case 0:

					strcpy(Process[PROC_AVC].Name , "AVC");

					strcpy(VectorStateMach[VECT_AVC].Name , "AVC");

					AVC_Param_Set[i].pPrc = &Process[PROC_AVC];
					AVC_Param_Set[i].pVect = &VectorStateMach[VECT_AVC];
					AVC_Param_Set[i].VectStateNum = 1;
					AVC_Param_Set[i].Mode = 0;

					AVC_Param_Set[i].MaxSpeedJog = 24.0;

					m->pCalib->Points[CALIB_TIG_VOLT_FBK].num = 10;
					AVC_Param_Set[i].pCalibPoints		= &m->pCalib->Points[CALIB_TIG_VOLT_FBK];

				break;

			}
		}

		for(i=0 ; i < 1 ; i++){

			switch(i){

				case 0:

					strcpy(Process[PROC_OSC].Name , "OSC");
					strcpy(VectorStateMach[VECT_OSC].Name , "OSC");

					OSC_TML_Param_Set[i].pPrc = &Process[PROC_OSC];
					OSC_TML_Param_Set[i].pVect = &VectorStateMach[VECT_OSC];
					OSC_TML_Param_Set[i].VectStateNum = 1;
					OSC_TML_Param_Set[i].pTML = &TML_MTR_INST[TML_AX_OSC] ;

					OSC_TML_Param_Set[i].Mode = 0;

					////  New Oscillation concept - BEMF
					OSC_TML_Param_Set[i].mm2ticks = TML_MTR_INST[TML_AX_OSC]._cfg.units * TML_MTR_INST[TML_AX_OSC]._cfg.rev_scale;
			 		OSC_TML_Param_Set[i].SpeedFactor = 410;
					//OSC_TML_Param_Set[i].MaxOscAmpl = 1.0 * 25.4;
					OSC_TML_Param_Set[i].MaxOscAmpl = 0.0;

					/////////////////////////
					/////   Hardcoded Limits
					if(cfg->HeadCfg.OSC.Limits_Harcoded){

						curCalib->Points[CALIB_OSC_SFT_LIMIT].num = 4;
						curCalib->Points[CALIB_OSC_SFT_LIMIT].val[0] = 10.0;
						curCalib->Points[CALIB_OSC_SFT_LIMIT].val[1] = 75.0;
						curCalib->Points[CALIB_OSC_SFT_LIMIT].val[2] = curCalib->Points[i].val[0];
						curCalib->Points[CALIB_OSC_SFT_LIMIT].val[3] = curCalib->Points[i].val[1];
					}

					////////////////////////////////////////////////

				break;

			}

		}

		for(i=0 ; i < 1 ; i++){

			switch(i){

				case 0:

					strcpy(Process[PROC_GAS].Name , "GAS");
					GAS_Param_Set[i].pPrc = &Process[PROC_GAS];

					//GAS_Param_Set[i].pSensInput     = &Hardware[1].Inp[5];  //FourAxis Head
					GAS_Param_Set[i].pOutput		= &Hardware[1].Outp[4];

				break;

			}

		}

		for(i=0 ; i < 1; i++){

			switch(i){

				case 0:

					strcpy(Process[PROC_COOL].Name , "COOLANT");
					COOL_Param_Set[i].pPrc = &Process[PROC_COOL];

					COOL_Param_Set[i].pSensInput     = &Hardware[1].Inp[4];  //FourAxis Head
					COOL_Param_Set[i].pOutput		= &Hardware[1].Outp[6];

				break;

			}

		}

		for(i=0 ; i < 1; i++){

			switch(i){

				case 0:

					strcpy(Process[PROC_HW_PS].Name , "HW PS");
					HW_PS_Param_Set[i].pPrc = &Process[PROC_HW_PS];

					HW_PS_Param_Set[i].pCalibPoints		= &m->pCalib->Points[CALIB_HW_AMPS_CMD];
					HW_PS_Param_Set[i].rawCmdMax 		= 16383.0;
					HW_PS_Param_Set[i].AmpCMD_Max 		= 160.0;

				break;

			}

		}

		for(i=0 ; i < 2; i++){

			switch(i){

				case 0:

					strcpy(Process[PROC_WIRE_FEED].Name ,"WrFeed");
					strcpy(VectorStateMach[VECT_WF].Name ,"WrFeed#1");
					strcpy(VectorStateMach[VECT_WF_1].Name ,"WrFeed#2");

					WIRE_Param_Set[i].pPrc = &Process[PROC_WIRE_FEED];
					WIRE_Param_Set[i].pVect = &VectorStateMach[m->pCfg->HeadCfg.WF.VECT_A_Indx];
					WIRE_Param_Set[i].VectStateNum = 1;
					WIRE_Param_Set[i].Mode = 0;  // classic

					WIRE_Param_Set[i].pCalibPoints	= &m->pCalib->Points[CALIB_WF_SPEED_CMD];

				break;

				case 1:

					strcpy(Process[PROC_WIRE_PULSE].Name ,"WrPulse");
					strcpy(VectorStateMach[VECT_WP].Name ,"WrPulse#1");
					strcpy(VectorStateMach[VECT_WP_1].Name ,"WrPulse#2");

					WIRE_Param_Set[i].pPrc = &Process[PROC_WIRE_PULSE];
					WIRE_Param_Set[i].pVect = &VectorStateMach[m->pCfg->HeadCfg.WP.VECT_A_Indx];
					WIRE_Param_Set[i].VectStateNum = 1;

					WIRE_Param_Set[i].pCalibPoints	= &m->pCalib->Points[CALIB_WP_SPEED_CMD];

				break;

		}

		}

		for(i=0 ; i < 1; i++){

			switch(i){

				case 0:

					strcpy(Process[PROC_TVL].Name , "TVL");
					strcpy(VectorStateMach[VECT_TVL].Name , "TVL");

					TVL_ROT_Param_Set[i].pPrc = &Process[PROC_TVL];
					TVL_ROT_Param_Set[i].pVect = &VectorStateMach[VECT_TVL];
					TVL_ROT_Param_Set[i].VectStateNum = 1;

					TVL_ROT_Param_Set[i].VectModeForJog = vectSt_Mode_Volt;

					TVL_ROT_Param_Set[i].MaxSpeedJog = 24.0;

					TVL_ROT_Param_Set[i].TotalRescaleFactor = 1.0;
					TVL_ROT_Param_Set[i].pCalibPoints = &m->pCalib->Points[CALIB_TVL_SPEED_CMD];

					TVL_ROT_Param_Set[i].pTrackDia = &curCfg->Param[parTVL_TrackDia].val[0];
					TVL_ROT_Param_Set[i].pVelTolerance = &curCfg->Param[parTVL_SpeedTolerane].val[0];

					TVL_ROT_Param_Set[i].pEncoder = &AxisCh[TML_AX_TVL].curPos;
					TVL_ROT_Param_Set[i].pHomePos = &OLD_MTR_POS[TVL_ENC_HOME];
					TVL_ROT_Param_Set[i].EncPerTick = m->pCfg->HeadCfg.TVL.EncPerTick;
					TVL_ROT_Param_Set[i].EncDir = m->pCfg->HeadCfg.TVL.Enc_Dir;
					TVL_ROT_Param_Set[i].TicksAtHighVel = 3;

				break;

			}
		}

		for(i=0 ; i < 1 ; i++){

			switch(i){

				case 0:

					strcpy(Process[m->pCfg->HeadCfg.INDX.PROC_Indx].Name , "INDX");
					INDEX_Param_Set[i].pPrc = &Process[m->pCfg->HeadCfg.INDX.PROC_Indx];
					Process[m->pCfg->HeadCfg.INDX.PROC_Indx].Disable = 1;

				break;

			}

		}

	return 1;

}

DINT Configure_U_BEND_HP_ENC_BEMF(MASTER_typ * m,UINT headType){
int i;

CurCfg_typ *curCfg;
Cfg_typ *cfg;
CurCalib_typ *curCalib , *defaultCalib;

	if(!m)
		return;

	curCfg = (CurCfg_typ*)m->pCurCfg;
	cfg = (Cfg_typ*)m->pCfg;

	curCalib = m->pCalib;
	defaultCalib = m->pDefaultCalib;

	if(!curCfg || !cfg || !curCalib  || !defaultCalib)
		return;

	/*********************************************/
	/***   Hardware and Vectors *********************/

	TML_MTR_INST[m->pCfg->HeadCfg.TVL.TML_Indx ].pState = &VectorStateMach[m->pCfg->HeadCfg.TVL.VECT_Indx];

	TML_MTR_INST[m->pCfg->HeadCfg.AVC.TML_A_Indx ].pState = &VectorStateMach[m->pCfg->HeadCfg.AVC.VECT_A_Indx];
	TML_MTR_INST[m->pCfg->HeadCfg.AVC.TML_B_Indx ].pState = &VectorStateMach[m->pCfg->HeadCfg.AVC.VECT_B_Indx];

	TML_MTR_INST[m->pCfg->HeadCfg.OSC.TML_A_Indx ].pState = &VectorStateMach[m->pCfg->HeadCfg.OSC.VECT_A_Indx];
	TML_MTR_INST[m->pCfg->HeadCfg.OSC.TML_B_Indx ].pState = &VectorStateMach[m->pCfg->HeadCfg.OSC.VECT_B_Indx];

	DC_Mtr[m->pCfg->HeadCfg.WF.DC_A_Indx ].pState = &VectorStateMach[m->pCfg->HeadCfg.WF.VECT_A_Indx];
	DC_Mtr[m->pCfg->HeadCfg.WP.DC_A_Indx ].pState = &VectorStateMach[m->pCfg->HeadCfg.WP.VECT_A_Indx];
	DC_Mtr[m->pCfg->HeadCfg.WF.DC_B_Indx ].pState = &VectorStateMach[m->pCfg->HeadCfg.WF.VECT_B_Indx];
	DC_Mtr[m->pCfg->HeadCfg.WP.DC_B_Indx ].pState = &VectorStateMach[m->pCfg->HeadCfg.WP.VECT_B_Indx];

/*

	VectorStateMach[VECT_AVC].simul = 1;
	VectorStateMach[VECT_OSC].simul = 1;
	VectorStateMach[VECT_TVL].simul = 1;
	VectorStateMach[VECT_WF].simul = 1;
	VectorStateMach[VECT_WP].simul = 1;
	VectorStateMach[VECT_WF_1].simul = 1;
	VectorStateMach[VECT_WP_1].simul = 1;
		m->pCfg->HeadCfg.WF.VECT_A_Indx]
	DC_Mtr[DC_AX_WF].Disable = 1;
	DC_Mtr[DC_AX_WP].Disable = 1;
	DC_Mtr[DC_AX_WF_1].Disable = 1;
	DC_Mtr[DC_AX_WP_1].Disable = 1;

	TML_MTR_INST[TML_AX_AVC].Disable = 1;
	TML_MTR_INST[TML_AX_OSC].Disable = 1;
	TML_MTR_INST[TML_AX_TVL].Disable = 1;

	//Process[PROC_AVC].Disable = 1;
	Process[PROC_AVC].TestMode = 1;
*/
	Process[PROC_TVL].Disable = 0;
	Process[PROC_OSC].Disable = 0;
	Process[PROC_AVC].Disable = 0;
	Process[PROC_WIRE_FEED].Disable = 0;
	Process[PROC_WIRE_PULSE].Disable = 0;

	VectorStateMach[VECT_AVC].simul = 0;
	VectorStateMach[VECT_OSC].simul = 0;
	VectorStateMach[VECT_TVL].simul = 0;

	VectorStateMach[VECT_WF].simul 		= 0;
	VectorStateMach[VECT_WF_1].simul 	= 0;
	VectorStateMach[VECT_WP].simul 		= 0;
	VectorStateMach[VECT_WP_1].simul 	= 0;

	DC_Mtr[DC_AX_WF].Disable = 0;
	DC_Mtr[DC_AX_WP].Disable = 0;
	DC_Mtr[DC_AX_WF_1].Disable = 0;
	DC_Mtr[DC_AX_WP_1].Disable = 0;

	TML_MTR_INST[TML_AX_AVC].Disable = 0;
	TML_MTR_INST[TML_AX_OSC].Disable = 0;
	TML_MTR_INST[TML_AX_TVL].Disable = 0;

	/*********************************************************/
	/****   Phisical hardware configuration   ************************/

		for(i = 0 ; i < PROCESS_NUM; i++)
			strcpy(Process[i].Name , "spare");

		for(i = 0 ; i < VECTORS_NUM; i++)
			strcpy(VectorStateMach[i].Name , "spare");

		//////////////////////////////////////////////////////////////////////////////////
		// Wire Block
		for(i=0 ; i < 2; i++){

			switch(i){

				case 0:
					strcpy(Process[m->pCfg->HeadCfg.WB[i].PROC_Indx].Name , "WB_UD");
					strcpy(VectorStateMach[m->pCfg->HeadCfg.WB[i].VECT_Indx].Name , "WB_UD");

					WR_BLK_Param_Set[i].pPrc = &Process[m->pCfg->HeadCfg.WB[i].PROC_Indx];
					WR_BLK_Param_Set[i].pVect = &VectorStateMach[m->pCfg->HeadCfg.WB[i].VECT_Indx];
					WR_BLK_Param_Set[i].VectStateNum = 1;

					WR_BLK_Param_Set[i].MaxSpeedJog = 24.0;

					Gen_one = 1.0;
					WR_BLK_Param_Set[i].pJogSpeed = &Gen_one;

				break;

				case 1:
					strcpy(Process[m->pCfg->HeadCfg.WB[i].PROC_Indx].Name , "WB_LR");
					strcpy(VectorStateMach[m->pCfg->HeadCfg.WB[i].VECT_Indx].Name , "WB_LR");

					WR_BLK_Param_Set[i].pPrc = &Process[PROC_WB_LR];
					WR_BLK_Param_Set[i].pVect = &VectorStateMach[VECT_WB_LR];
					WR_BLK_Param_Set[i].VectStateNum = 1;

					WR_BLK_Param_Set[i].MaxSpeedJog = 24.0;

					Gen_one = 1.0;
					WR_BLK_Param_Set[i].pJogSpeed = &Gen_one;

				break;

			}

		}

		for(i = 0 ; i < DC2DIRMTR_NUM; i++){

			switch(i){

				case DC_WB_UD:

					strcpy(DC2DirMtr[i].Name , "WB_UD");
					DC2DirMtr[i].pState = &VectorStateMach[VECT_WB_UD];

					DC2DirMtr[i].Cfg.pQ1_output = &Hardware[1].Outp[12];
					DC2DirMtr[i].Cfg.pQ2_output = &Hardware[1].Outp[13];
					DC2DirMtr[i].Cfg.pQ3_output = &Hardware[1].Outp[14];
					DC2DirMtr[i].Cfg.pQ4_output = &Hardware[1].Outp[15];

					DC2DirMtr[i].Cfg.MtrDir = 1.0;

				break;

				case DC_WB_LR:

					strcpy(DC2DirMtr[i].Name , "WB_LR");
					DC2DirMtr[i].pState = &VectorStateMach[VECT_WB_LR];

					DC2DirMtr[i].Cfg.pQ1_output = &Hardware[1].Outp[16];
					DC2DirMtr[i].Cfg.pQ2_output = &Hardware[1].Outp[17];
					DC2DirMtr[i].Cfg.pQ3_output = &Hardware[1].Outp[18];
					DC2DirMtr[i].Cfg.pQ4_output = &Hardware[1].Outp[19];

					DC2DirMtr[i].Cfg.MtrDir = 1.0;

				break;

			}

		}
		/////////////////////////////////////////////////////////////////////////////////

		for(i = 0 ; i < GEN_MTR_NUM; i++){

			switch(i){

				case DC_AX_WF:
				case DC_AX_WF_1:

					switch(i){

						case DC_AX_WF:

							strcpy(DC_Mtr[i].Name , "DC WFeed#1");

							DC_Mtr[i].Cfg.mtr_dir = -1.0;

							if(ProjectConfig == project_US_Orbital) // US Orbital has B and /B swapped
								DC_Mtr[i].Cfg.enc_dir = -1.0;
							else
								DC_Mtr[i].Cfg.enc_dir = 1.0;

						break;

						case DC_AX_WF_1:

							strcpy(DC_Mtr[i].Name , "DC WFeed#2");

							DC_Mtr[i].Cfg.mtr_dir = 1.0;

							if(ProjectConfig == project_US_Orbital) // US Orbital has B and /B swapped
								DC_Mtr[i].Cfg.enc_dir = -1.0;
							else
								DC_Mtr[i].Cfg.enc_dir = 1.0;

						break;

					}

					//DC_Mtr[i].Cfg.units = 59.847340050885561192713356451475; // 0.75 " dia * 25.4 * PI
					DC_Mtr[i].Cfg.units = 2000 / 59.847340050885561192713356451475; // 2000 enc ticks / 0.75 " dia * 25.4 * PI
					DC_Mtr[i].Cfg.rev_scale = 66.0;	// Ratio gear box 66:1

					/* Parameters for PID controller */
					// To nowe
					DC_Mtr[i].msc.PIDParameters.Kp= 1.0;//0.4; //proportional gain / was 0.6
					//DC_Mtr[i].msc.PIDParameters.Kp= 0.1;//0.4; //proportional gain / was 0.6
					DC_Mtr[i].msc.PIDParameters.Tn= 0.1;//0.3.1; //intergral action time
					DC_Mtr[i].msc.PIDParameters.Kfbk = 0.01; //windup dampenin

					DC_Mtr[i].msc.PID.enable = 0;
					DC_Mtr[i].msc.PID.pPar = &DC_Mtr[i].msc.PIDParameters;
					DC_Mtr[i].msc.PID.request = 3; // Read parameters from PIDParameters
					DC_Mtr[i].msc.PIDParameters.Tv= 0; //derivative action time
					DC_Mtr[i].msc.PIDParameters.Y_max = 100.0;  //max manipulated variable %
					DC_Mtr[i].msc.PIDParameters.Y_min = -100.0; //min manipulated variable %

				break;

				case DC_AX_WP:
				case DC_AX_WP_1:

					switch(i){

						case DC_AX_WP:

							strcpy(DC_Mtr[i].Name , "DC WPulse#1");

							DC_Mtr[i].Cfg.mtr_dir = 1.0;

							if(ProjectConfig == project_US_Orbital) // US Orbital has B and /B swapped
								DC_Mtr[i].Cfg.enc_dir = -1.0;
							else
								DC_Mtr[i].Cfg.enc_dir = 1.0;

						break;

						case DC_AX_WP_1:

							strcpy(DC_Mtr[i].Name , "DC WPulse#2");

							DC_Mtr[i].Cfg.mtr_dir = 1.0;

							if(ProjectConfig == project_US_Orbital) // US Orbital has B and /B swapped
								DC_Mtr[i].Cfg.enc_dir = -1.0;
							else
								DC_Mtr[i].Cfg.enc_dir = 1.0;

						break;

					}

					//oryginalnie jest 2000 pulsow na obrot potem ratio on gear 4.8 : 1
					DC_Mtr[i].Cfg.units = 2000;
					DC_Mtr[i].Cfg.rev_scale = 4.8;// ratio on gear 4.8

					/* Parameters for PID controller */
					// To nowe
					DC_Mtr[i].msc.PIDParameters.Kp= 1.0;//0.4; //proportional gain / was 0.6
					//DC_Mtr[i].msc.PIDParameters.Kp= 0.1;//0.4; //proportional gain / was 0.6
					DC_Mtr[i].msc.PIDParameters.Tn= 0.1;//0.3.1; //intergral action time
					DC_Mtr[i].msc.PIDParameters.Kfbk = 0.01; //windup dampenin

					DC_Mtr[i].msc.PID.enable = 0;
					DC_Mtr[i].msc.PID.pPar = &DC_Mtr[i].msc.PIDParameters;
					DC_Mtr[i].msc.PID.request = 3; // Read parameters from PIDParameters
					DC_Mtr[i].msc.PIDParameters.Tv= 0; //derivative action time
					DC_Mtr[i].msc.PIDParameters.Y_max = 100.0;  //max manipulated variable %
					DC_Mtr[i].msc.PIDParameters.Y_min = -100.0; //min manipulated variable %

				break;

				default:

					//strcpy(DC_Mtr[i].Name , "Spare ");
					xsprintf(DC_Mtr[i].Name, "Spare %d", i );

				break;

			}

			//CalcUnits(&DC_Mtr[i]);
			DC_Mtr[i].msc.kPos = (float)DC_Mtr[i].Cfg.units * DC_Mtr[i].Cfg.rev_scale;

		}

		/***********************************/

			for(i = 0 ; i < TML_SERVO_NUM ; i++){

				switch(i){

					// tml->_int.kPos = (tml->_cfg.units * tml->_cfg.rev_scale) / tml->_cfg.rev_motor;
					case TML_AX_AVC:

						strcpy(TML_MTR_INST[i].Name , "AVC");

						// Analog Feedback from REF
						//TML_MTR_INST[i]._cfg.loopPeriod = 0.001;
						TML_MTR_INST[i]._cfg.units = 4095;
						//TML_MTR_INST[i]._cfg.rev_motor = 1;
						TML_MTR_INST[i]._cfg.rev_scale = 1.0/5.0;
						//TML_MTR_INST[i]._cfg.maxVel = 10.0; //1//6000 rpm
						//TML_MTR_INST[i]._cfg.maxAcc = 100000.0;
						//TML_MTR_INST[i]._cfg.satpMax = 27853; // KPP bylo Stauration of proportional gain
						TML_MTR_INST[i]._cfg.satpMax = 32000; // KPP bylo Stauration of proportional gain
						//TML_MTR_INST[i]._cfg.kppMax = 32000; // KPP bylo Stauration of proportional gain
						//TML_MTR_INST[i]._cfg.kipMax = 200; // KPP bylo Stauration of proportional gain
						TML_MTR_INST[i]._cfg.absFbk = 0; // absolute value feedback

						TML_MTR_INST[i]._cfg.signFilter = curCfg->Param[parAVC_FbkFilter].val[0];

						if(ProjectConfig == project_US_Orbital){
							strcpy(TML_MTR_INST[i]._cfg.programName , "1123_AVC_U_BEND_ENC_US_BEMF.sw");
							TML_MTR_INST[i].ProgramVersion = ASC2UDINT("1123");
							TML_MTR_INST[i].FirmwareVersion = ASC2UDINT("6A2B");  //0x674B
							TML_MTR_INST[i]._cfg.Appl_ID_adr = 0x7FCF;
							TML_MTR_INST[i]._cfg.rev_motor = -1.0;
							TML_MTR_INST[i]._cfg.kppMax = -32000; // KPP bylo Stauration of proportional gain
							TML_MTR_INST[i]._cfg.kipMax = -200; // KPP bylo Stauration of proportional gain

							TML_MTR_INST[i]._cfg.maxVel = 200.0; //1//6000 rpm
							TML_MTR_INST[i]._cfg.maxAcc = 100000.0;

							TML_MTR_INST[i]._cfg.loopPeriod = 0.01; // real BEMF - experimental value

						}
						else{
							strcpy(TML_MTR_INST[i]._cfg.programName , "0023_AVC_U_BEND_ENC.sw");
							TML_MTR_INST[i].ProgramVersion = ASC2UDINT("0023");
							TML_MTR_INST[i].FirmwareVersion = ASC2UDINT("674C");  //0x674C
							TML_MTR_INST[i]._cfg.rev_motor = 1.0;
							TML_MTR_INST[i]._cfg.kppMax = 32000; // KPP bylo Stauration of proportional gain
							TML_MTR_INST[i]._cfg.kipMax = 200; // KPP bylo Stauration of proportional gain

							TML_MTR_INST[i]._cfg.maxVel = 10.0; //1//6000 rpm
							TML_MTR_INST[i]._cfg.maxAcc = 100000.0;

							TML_MTR_INST[i]._cfg.loopPeriod = 0.001;
						}

						//TML_MTR_INST[i]._cfg.sftLimitPos = 1000.0;
						//TML_MTR_INST[i]._cfg.sftLimitNeg = -1000.0;

					break;

					case TML_AX_OSC:

						strcpy(TML_MTR_INST[i].Name , "OSC");

						if(ProjectConfig == project_US_Orbital){
							strcpy(TML_MTR_INST[i]._cfg.programName , "1122_OSC_U_BEND_ENC_US_BEMF.sw");
							TML_MTR_INST[i].ProgramVersion = ASC2UDINT("1122");
							TML_MTR_INST[i].FirmwareVersion = ASC2UDINT("6A2B");  //0x674B
							TML_MTR_INST[i]._cfg.Appl_ID_adr = 0x7FCF;
							//TML_MTR_INST[i]._cfg.rev_motor = -1.0;
							TML_MTR_INST[i]._cfg.rev_motor = 1.0;

						}
						else{
							strcpy(TML_MTR_INST[i]._cfg.programName , "0022_OSC_U_BEND_ENC.sw");
							TML_MTR_INST[i].ProgramVersion = ASC2UDINT("0022");
							TML_MTR_INST[i].FirmwareVersion = ASC2UDINT("674C");  //0x674C
							TML_MTR_INST[i]._cfg.rev_motor = 1.0;

						}

						TML_MTR_INST[i]._cfg.loopPeriod = 0.001;
						TML_MTR_INST[i]._cfg.absFbk = 0; // value fom APOS which is analog Ref
						TML_MTR_INST[i]._cfg.units = 4096.0 ;
						//TML_MTR_INST[i]._cfg.rev_motor = 1;
						TML_MTR_INST[i]._cfg.rev_scale = 1.0 / 80.0;  // this comes from experiment
						//TML_MTR_INST[i]._cfg.rev_scale = 1.0 / 56.0; // this comes from drawings
						TML_MTR_INST[i]._cfg.maxVel = 100.0;
						TML_MTR_INST[i]._cfg.maxAcc = 100.0;

						TML_MTR_INST[i]._cfg.AnalLimitPos = 3900;
						TML_MTR_INST[i]._cfg.AnalLimitNeg = 100;

					break;

					case TML_AX_TVL:

						strcpy(TML_MTR_INST[i].Name , "TVL");

						/// Deferent TML programs
						// Back EMF
						TML_MTR_INST[i]._cfg.loopPeriod = 0.001;

						if(ProjectConfig == project_US_Orbital){

							strcpy(TML_MTR_INST[i]._cfg.programName , "1021_TVL_U_BEND_ENC_US.sw");
							TML_MTR_INST[i].ProgramVersion = ASC2UDINT("1021");
							TML_MTR_INST[i].FirmwareVersion = ASC2UDINT("6A2B");  //0x674B
							TML_MTR_INST[i]._cfg.Appl_ID_adr = 0x7FCF;
							TML_MTR_INST[i]._cfg.rev_motor = -1.0;
							TML_MTR_INST[i]._cfg.rev_scale = -1920.0;
							TML_MTR_INST[i]._cfg.units =  1000; //  to jest tyle ile z max speed TML EREF

							/* gotowe
							strcpy(TML_MTR_INST[i]._cfg.programName , "1121_TVL_U_BEND_ENC_US_BEMF.sw");
							TML_MTR_INST[i].ProgramVersion = ASC2UDINT("1121");
							TML_MTR_INST[i].FirmwareVersion = ASC2UDINT("6A2B");  //0x674B
							TML_MTR_INST[i]._cfg.Appl_ID_adr = 0x7FCF;
							TML_MTR_INST[i]._cfg.rev_motor = -1.0;
							TML_MTR_INST[i]._cfg.rev_scale = -1920.0;
							TML_MTR_INST[i]._cfg.units =  70;
							*/

						}
						else{
							strcpy(TML_MTR_INST[i]._cfg.programName , " 1021_TVL_U_BEND_ENC_US.sw");
							TML_MTR_INST[i].ProgramVersion = ASC2UDINT("1021");
							TML_MTR_INST[i].FirmwareVersion = ASC2UDINT("674C");  //0x674C
							TML_MTR_INST[i]._cfg.rev_motor = -1.0;
							TML_MTR_INST[i]._cfg.rev_scale = -1920.0;
							TML_MTR_INST[i]._cfg.units =  1000; //  to jest tyle ile z max speed TML EREF
						}

						//TML_MTR_INST[i]._cfg.rev_scale = -1920.0;
						//TML_MTR_INST[i]._cfg.rev_motor = 1.0 ;
						TML_MTR_INST[i]._cfg.maxVel =  10.0; // mm/s
						TML_MTR_INST[i]._cfg.maxAcc = 100.0;
						TML_MTR_INST[i]._cfg.absFbk = 0; // non absolute value feedback , remember last value before drive reset

					break;

					default:

						//xsprintf(TML_MTR_INST[i].Name, "Spare %d", i );
						xsprintf(TML_MTR_INST[i].Name, "Spare %d", i );

					break;

				}

			TML_MTR_INST[i].xCMD = TML_RESTART;

		}

		TML_mgr[0].hrdw[0].AxisNum = 3;
		TML_mgr[0].hrdw[1].AxisNum = 0;

		TML_mgr[0].pAxis[0] = &AxisCh[0];
		TML_mgr[0].pAxis[1] = 0;
		//TML_mgr[0].pAxis[1] = &AxisCh[TML_mgr[0].hrdw[0].AxisNum];

		TML_mgr[0].pTML[0] = &TML_MTR_INST[0];
		TML_mgr[0].pTML[1] = 0;
		//TML_mgr[0].pTML[1] = &TML_MTR_INST[TML_mgr[0].hrdw[0].AxisNum];

		AxisCh[TML_AX_TVL].AxisID	= 1;
		AxisCh[TML_AX_OSC].AxisID 	= 2;
		AxisCh[TML_AX_AVC].AxisID 	= 3;

		/**************************************/
		/****   Process   ************************/

		// Lincoln Power Supply
		for(i=0 ; i < 1; i++){

			switch(i){

				case 0:

					strcpy(Process[PROC_TIG_PS].Name , "TIG PS");
					PS_Param_Set[i].pPrc = &Process[PROC_TIG_PS];

					PS_Param_Set[i].pCalibPoints		= &m->pCalib->Points[CALIB_TIG_AMPS_CMD];
					//PS_Param_Set[i].rawCmdMax			= 26170; // //
					//PS_Param_Set[i].AmpCMD_Max			= 500.0; // 62.5 amp / 1 V
					PS_Param_Set[i].rawCmdMax			= 32767;
					PS_Param_Set[i].AmpCMD_Max			= 627.0;

					PS_Param_Set[i].pArcLinkRobot   = (UDINT)&ArcLink.robot;

				break;

			}

		}

		for(i=0 ; i < 1 ; i++){

			switch(i){

				case 0:

					strcpy(Process[PROC_AVC].Name , "AVC");

					strcpy(VectorStateMach[VECT_AVC].Name , "AVC");

					AVC_Param_Set[i].pPrc = &Process[PROC_AVC];
					AVC_Param_Set[i].pVect = &VectorStateMach[VECT_AVC];
					AVC_Param_Set[i].VectStateNum = 1;
					AVC_Param_Set[i].Mode = 2; // Real BEMF Speed control

					AVC_Param_Set[i].MaxSpeedJog = 24.0;

					if(ProjectConfig == project_US_Orbital){
						AVC_Param_Set[i].maxBEMFspeed = 200.0;
						AVC_Param_Set[i].Mode = 2; // Real BEMF Speed control
					}
					else{

						AVC_Param_Set[i].Mode = 0;

					}

					m->pCalib->Points[CALIB_TIG_VOLT_FBK].num = 10;
					AVC_Param_Set[i].pCalibPoints		= &m->pCalib->Points[CALIB_TIG_VOLT_FBK];

				break;

			}
		}

		for(i=0 ; i < 1 ; i++){

			switch(i){

				case 0:

					strcpy(Process[PROC_OSC].Name , "OSC");
					strcpy(VectorStateMach[VECT_OSC].Name , "OSC");

					OSC_TML_Param_Set[i].pPrc = &Process[PROC_OSC];
					OSC_TML_Param_Set[i].pVect = &VectorStateMach[VECT_OSC];
					OSC_TML_Param_Set[i].VectStateNum = 1;
					OSC_TML_Param_Set[i].pTML = &TML_MTR_INST[TML_AX_OSC] ;

					OSC_TML_Param_Set[i].Mode = 0;

					////  New Oscillation concept - BEMF
					OSC_TML_Param_Set[i].mm2ticks = TML_MTR_INST[TML_AX_OSC]._cfg.units * TML_MTR_INST[TML_AX_OSC]._cfg.rev_scale;
			 		//OSC_TML_Param_Set[i].SpeedFactor = 410;
					//OSC_TML_Param_Set[i].MaxOscAmpl = 1.0 * 25.4;
					OSC_TML_Param_Set[i].MaxOscAmpl = 0.0;

					if(ProjectConfig == project_US_Orbital)
						OSC_TML_Param_Set[i].SpeedFactor = 100; // Real BEMF
					else
						OSC_TML_Param_Set[i].SpeedFactor = 410;

					/////////////////////////
					/////   Hardcoded Limits
					if(cfg->HeadCfg.OSC.Limits_Harcoded){

						curCalib->Points[CALIB_OSC_SFT_LIMIT].num = 4;
						curCalib->Points[CALIB_OSC_SFT_LIMIT].val[0] = 10.0;
						curCalib->Points[CALIB_OSC_SFT_LIMIT].val[1] = 75.0;
						curCalib->Points[CALIB_OSC_SFT_LIMIT].val[2] = curCalib->Points[i].val[0];
						curCalib->Points[CALIB_OSC_SFT_LIMIT].val[3] = curCalib->Points[i].val[1];
					}

					////////////////////////////////////////////////

				break;

			}

		}

		for(i=0 ; i < 1 ; i++){

			switch(i){

				case 0:

					strcpy(Process[PROC_GAS].Name , "GAS");
					GAS_Param_Set[i].pPrc = &Process[PROC_GAS];

					//GAS_Param_Set[i].pSensInput     = &Hardware[1].Inp[5];  //FourAxis Head
					GAS_Param_Set[i].pOutput		= &Hardware[1].Outp[4];

				break;

			}

		}

		for(i=0 ; i < 1; i++){

			switch(i){

				case 0:

					strcpy(Process[PROC_COOL].Name , "COOLANT");
					COOL_Param_Set[i].pPrc = &Process[PROC_COOL];

					COOL_Param_Set[i].pSensInput     = &Hardware[1].Inp[4];  //FourAxis Head
					COOL_Param_Set[i].pOutput		= &Hardware[1].Outp[6];

				break;

			}

		}

		for(i=0 ; i < 1; i++){

			switch(i){

				case 0:

					strcpy(Process[PROC_HW_PS].Name , "HW PS");
					HW_PS_Param_Set[i].pPrc = &Process[PROC_HW_PS];

					HW_PS_Param_Set[i].pCalibPoints		= &m->pCalib->Points[CALIB_HW_AMPS_CMD];
					HW_PS_Param_Set[i].rawCmdMax 		= 16383.0;
					HW_PS_Param_Set[i].AmpCMD_Max 		= 160.0;

				break;

			}

		}

		for(i=0 ; i < 2; i++){

			switch(i){

				case 0:

					strcpy(Process[PROC_WIRE_FEED].Name ,"WrFeed");
					strcpy(VectorStateMach[VECT_WF].Name ,"WrFeed#1");
					strcpy(VectorStateMach[VECT_WF_1].Name ,"WrFeed#2");

					WIRE_Param_Set[i].pPrc = &Process[PROC_WIRE_FEED];
					WIRE_Param_Set[i].pVect = &VectorStateMach[m->pCfg->HeadCfg.WF.VECT_A_Indx];
					WIRE_Param_Set[i].VectStateNum = 1;
					WIRE_Param_Set[i].Mode = 0;  // classic

					WIRE_Param_Set[i].pCalibPoints	= &m->pCalib->Points[CALIB_WF_SPEED_CMD];

				break;

				case 1:

					strcpy(Process[PROC_WIRE_PULSE].Name ,"WrPulse");
					strcpy(VectorStateMach[VECT_WP].Name ,"WrPulse#1");
					strcpy(VectorStateMach[VECT_WP_1].Name ,"WrPulse#2");

					WIRE_Param_Set[i].pPrc = &Process[PROC_WIRE_PULSE];
					WIRE_Param_Set[i].pVect = &VectorStateMach[m->pCfg->HeadCfg.WP.VECT_A_Indx];
					WIRE_Param_Set[i].VectStateNum = 1;

					WIRE_Param_Set[i].pCalibPoints	= &m->pCalib->Points[CALIB_WP_SPEED_CMD];

				break;

		}

		}

		for(i=0 ; i < 1; i++){

			switch(i){

				case 0:

					strcpy(Process[PROC_TVL].Name , "TVL");
					strcpy(VectorStateMach[VECT_TVL].Name , "TVL");

					TVL_ROT_Param_Set[i].pPrc = &Process[PROC_TVL];
					TVL_ROT_Param_Set[i].pVect = &VectorStateMach[VECT_TVL];
					TVL_ROT_Param_Set[i].VectStateNum = 1;

					TVL_ROT_Param_Set[i].VectModeForJog = vectSt_Mode_Volt;
					//TVL_ROT_Param_Set[i].VectModeForJog = vectSt_Mode_Vel;

					TVL_ROT_Param_Set[i].MaxSpeedJog = 24.0;

					TVL_ROT_Param_Set[i].TotalRescaleFactor = 1.0;
					TVL_ROT_Param_Set[i].pCalibPoints = &m->pCalib->Points[CALIB_TVL_SPEED_CMD];

					TVL_ROT_Param_Set[i].pTrackDia = &curCfg->Param[parTVL_TrackDia].val[0];
					TVL_ROT_Param_Set[i].pVelTolerance = &curCfg->Param[parTVL_SpeedTolerane].val[0];
```
